LIN {X 0,Y 466.068,Z 1064.204,A -85,B 0,C 180,E1 20747.984,E2 20747.984} C_VEL
LIN {X 0,Y 471.463,Z 1046.564,A -85,B 0,C 180,E1 20746.009,E2 20746.009} C_VEL
LIN {X 0,Y 478.479,Z 1022.709,A -85,B 0,C 180,E1 20743.696,E2 20743.696} C_VEL
LIN {X 0,Y 484.027,Z 1002.948,A -85,B 0,C 180,E1 20742.045,E2 20742.045} C_VEL
LIN {X 0,Y 489.037,Z 984.19,A -85,B 0,C 180,E1 20740.666,E2 20740.666} C_VEL
LIN {X 0,Y 494.055,Z 964.129,A -85,B 0,C 180,E1 20739.369,E2 20739.369} C_VEL
LIN {X 0,Y 500.021,Z 937.929,A -85,B 0,C 180,E1 20737.922,E2 20737.922} C_VEL
LIN {X 0,Y 504.618,Z 915.146,A -85,B 0,C 180,E1 20736.878,E2 20736.878} C_VEL
LIN {X 0,Y 508.385,Z 894.221,A -85,B 0,C 180,E1 20736.067,E2 20736.067} C_VEL
LIN {X 0,Y 511.805,Z 872.432,A -85,B 0,C 180,E1 20735.363,E2 20735.363} C_VEL
LIN {X 0,Y 515.371,Z 845.255,A -85,B 0,C 180,E1 20734.667,E2 20734.667} C_VEL
LIN {X 0,Y 517.719,Z 818.939,A -85,B 0,C 180,E1 20734.166,E2 20734.166} C_VEL
LIN {X 0,Y 527.517,Z 618.648,A -85,B 0,C 180,E1 20731.083,E2 20731.083} C_VEL
LIN {X 0,Y 535.309,Z 463.056,A -85,B 0,C 180,E1 20728.673,E2 20728.673} C_VEL
LIN {X 0,Y 522.466,Z 443.048,A -85,B 0,C 180,E1 20726.054,E2 20726.054} C_VEL
LIN {X 0,Y 512.066,Z 427.582,A -85,B 0,C 180,E1 20723.719,E2 20723.719} C_VEL
LIN {X 0,Y 502.428,Z 413.843,A -85,B 0,C 180,E1 20721.327,E2 20721.327} C_VEL
LIN {X 0,Y 493.826,Z 402.221,A -85,B 0,C 180,E1 20718.964,E2 20718.964} C_VEL
LIN {X 0,Y 487.693,Z 394.13,A -85,B 0,C 180,E1 20717.11,E2 20717.11} C_VEL
LIN {X 0,Y 479.768,Z 384.005,A -85,B 0,C 180,E1 20714.421,E2 20714.421} C_VEL
LIN {X 0,Y 474.951,Z 378.127,A -85,B 0,C 180,E1 20712.585,E2 20712.585} C_VEL
LIN {X 0,Y 471.073,Z 373.273,A -85,B 0,C 180,E1 20710.951,E2 20710.951} C_VEL
LIN {X 0,Y 466.248,Z 367.542,A -85,B 0,C 180,E1 20708.66,E2 20708.66} C_VEL
LIN {X 0,Y 460.499,Z 361.075,A -85,B 0,C 180,E1 20705.357,E2 20705.357} C_VEL
LIN {X 0,Y 456.273,Z 356.326,A -85,B 0,C 180,E1 20702.21,E2 20702.21} C_VEL
LIN {X 0,Y 455.002,Z 354.829,A -85,B 0,C 180,E1 20701.007,E2 20701.007} C_VEL
LIN {X 0,Y 451.289,Z 351.259,A -85,B 0,C 180,E1 20695.17,E2 20695.17} C_VEL
LIN {X 0,Y 451.06,Z 350.914,A -85,B 0,C 180,E1 20691.972,E2 20691.972} C_VEL
LIN {X 0,Y 452.202,Z 352.442,A -85,B 0,C 180,E1 20688.133,E2 20688.133} C_VEL
LIN {X 0,Y 455.623,Z 355.438,A -85,B 0,C 180,E1 20683.948,E2 20683.948} C_VEL
LIN {X 0,Y 459.701,Z 360.404,A -85,B 0,C 180,E1 20680.694,E2 20680.694} C_VEL
LIN {X 0,Y 461.444,Z 362.203,A -85,B 0,C 180,E1 20679.582,E2 20679.582} C_VEL
LIN {X 0,Y 465.451,Z 366.813,A -85,B 0,C 180,E1 20677.319,E2 20677.319} C_VEL
LIN {X 0,Y 471.187,Z 373.665,A -85,B 0,C 180,E1 20674.55,E2 20674.55} C_VEL
LIN {X 0,Y 476.082,Z 379.677,A -85,B 0,C 180,E1 20672.514,E2 20672.514} C_VEL
LIN {X 0,Y 480.917,Z 385.697,A -85,B 0,C 180,E1 20670.717,E2 20670.717} C_VEL
LIN {X 0,Y 487.922,Z 394.605,A -85,B 0,C 180,E1 20668.392,E2 20668.392} C_VEL
LIN {X 0,Y 496.453,Z 405.98,A -85,B 0,C 180,E1 20665.88,E2 20665.88} C_VEL
LIN {X 0,Y 506.01,Z 419.292,A -85,B 0,C 180,E1 20663.362,E2 20663.362} C_VEL
LIN {X 0,Y 516.742,Z 435.021,A -85,B 0,C 180,E1 20660.819,E2 20660.819} C_VEL
LIN {X 0,Y 528.945,Z 454.078,A -85,B 0,C 180,E1 20658.214,E2 20658.214} C_VEL
LIN {X 0,Y 530.531,Z 456.882,A -85,B 0,C 180,E1 20657.888,E2 20657.888} C_VEL
LIN {X 0,Y 518.704,Z 687.315,A -85,B 0,C 180,E1 20654.4,E2 20654.4} C_VEL
LIN {X 0,Y 513.437,Z 790.124,A -85,B 0,C 180,E1 20652.825,E2 20652.825} C_VEL
LIN {X 0,Y 510.977,Z 817.179,A -85,B 0,C 180,E1 20652.266,E2 20652.266} C_VEL
LIN {X 0,Y 507.981,Z 840.872,A -85,B 0,C 180,E1 20651.597,E2 20651.597} C_VEL
LIN {X 0,Y 504.867,Z 861.286,A -85,B 0,C 180,E1 20650.884,E2 20650.884} C_VEL
LIN {X 0,Y 500.818,Z 884.029,A -85,B 0,C 180,E1 20649.93,E2 20649.93} C_VEL
LIN {X 0,Y 495.731,Z 908.011,A -85,B 0,C 180,E1 20648.7,E2 20648.7} C_VEL
LIN {X 0,Y 491.245,Z 926.964,A -85,B 0,C 180,E1 20647.56,E2 20647.56} C_VEL
LIN {X 0,Y 486.131,Z 946.852,A -85,B 0,C 180,E1 20646.178,E2 20646.178} C_VEL
LIN {X 0,Y 479.73,Z 969.616,A -85,B 0,C 180,E1 20644.317,E2 20644.317} C_VEL
LIN {X 0,Y 474.426,Z 987.14,A -85,B 0,C 180,E1 20642.651,E2 20642.651} C_VEL
LIN {X 0,Y 468.964,Z 1004.442,A -85,B 0,C 180,E1 20640.777,E2 20640.777} C_VEL
LIN {X 0,Y 462.391,Z 1024.359,A -85,B 0,C 180,E1 20638.265,E2 20638.265} C_VEL
LIN {X 0,Y 457.591,Z 1038.554,A -85,B 0,C 180,E1 20636.192,E2 20636.192} C_VEL
LIN {X 0,Y 453.023,Z 1052.055,A -85,B 0,C 180,E1 20633.96,E2 20633.96} C_VEL
LIN {X 0,Y 452.093,Z 1054.945,A -85,B 0,C 180,E1 20633.456,E2 20633.456} C_VEL
LIN {X 0,Y 449.768,Z 1059.456,A -85,B 0,C 180,E1 20632.709,E2 20632.709} C_VEL
LIN {X 0,Y 440.278,Z 1071.251,A -85,B 0,C 180,E1 20630.787,E2 20630.787} C_VEL
LIN {X 0,Y 438.47,Z 1074.724,A -85,B 0,C 180,E1 20630.085,E2 20630.085} C_VEL
LIN {X 0,Y 434.176,Z 1087.706,A -85,B 0,C 180,E1 20626.868,E2 20626.868} C_VEL
LIN {X 0,Y 431.232,Z 1097.26,A -85,B 0,C 180,E1 20624.09,E2 20624.09} C_VEL
LIN {X 0,Y 428.732,Z 1106.306,A -85,B 0,C 180,E1 20621.025,E2 20621.025} C_VEL
LIN {X 0,Y 426.702,Z 1114.7,A -85,B 0,C 180,E1 20617.54,E2 20617.54} C_VEL
LIN {X 0,Y 425.561,Z 1120.466,A -85,B 0,C 180,E1 20614.582,E2 20614.582} C_VEL
LIN {X 0,Y 424.864,Z 1124.898,A -85,B 0,C 180,E1 20611.753,E2 20611.753} C_VEL
LIN {X 0,Y 424.443,Z 1128.897,A -85,B 0,C 180,E1 20608.38,E2 20608.38} C_VEL
LIN {X 0,Y 424.242,Z 1131.291,A -85,B 0,C 180,E1 20604.997,E2 20604.997} C_VEL
LIN {X 0,Y 424.216,Z 1132.271,A -85,B 0,C 180,E1 20602.143,E2 20602.143} C_VEL
LIN {X 0,Y 424.205,Z 1132.282,A -85,B 0,C 180,E1 20599.393,E2 20599.393} C_VEL
LIN {X 0,Y 424.282,Z 1131.313,A -85,B 0,C 180,E1 20596.508,E2 20596.508} C_VEL
LIN {X 0,Y 424.543,Z 1128.64,A -85,B 0,C 180,E1 20592.879,E2 20592.879} C_VEL
LIN {X 0,Y 425.024,Z 1125,A -85,B 0,C 180,E1 20589.768,E2 20589.768} C_VEL
LIN {X 0,Y 425.805,Z 1120.621,A -85,B 0,C 180,E1 20586.912,E2 20586.912} C_VEL
LIN {X 0,Y 427.274,Z 1114.277,A -85,B 0,C 180,E1 20583.601,E2 20583.601} C_VEL
LIN {X 0,Y 429.569,Z 1105.855,A -85,B 0,C 180,E1 20580.125,E2 20580.125} C_VEL
LIN {X 0,Y 432.214,Z 1097.455,A -85,B 0,C 180,E1 20577.226,E2 20577.226} C_VEL
LIN {X 0,Y 435.991,Z 1086.706,A -85,B 0,C 180,E1 20574.05,E2 20574.05} C_VEL
LIN {X 0,Y 440.717,Z 1073.903,A -85,B 0,C 180,E1 20570.889,E2 20570.889} C_VEL
LIN {X 0,Y 445.319,Z 1062.002,A -85,B 0,C 180,E1 20568.349,E2 20568.349} C_VEL
LIN {X 0,Y 451.443,Z 1046.625,A -85,B 0,C 180,E1 20565.495,E2 20565.495} C_VEL
LIN {X 0,Y 457.914,Z 1030.027,A -85,B 0,C 180,E1 20562.898,E2 20562.898} C_VEL
LIN {X 0,Y 463.585,Z 1015.355,A -85,B 0,C 180,E1 20560.891,E2 20560.891} C_VEL
LIN {X 0,Y 470.718,Z 996.54,A -85,B 0,C 180,E1 20558.646,E2 20558.646} C_VEL
LIN {X 0,Y 477.551,Z 977.158,A -85,B 0,C 180,E1 20556.689,E2 20556.689} C_VEL
LIN {X 0,Y 483.256,Z 960.126,A -85,B 0,C 180,E1 20555.189,E2 20555.189} C_VEL
LIN {X 0,Y 488.91,Z 942.119,A -85,B 0,C 180,E1 20553.799,E2 20553.799} C_VEL
LIN {X 0,Y 495.538,Z 919.171,A -85,B 0,C 180,E1 20552.282,E2 20552.282} C_VEL
LIN {X 0,Y 500.941,Z 897.811,A -85,B 0,C 180,E1 20551.1,E2 20551.1} C_VEL
LIN {X 0,Y 505.444,Z 877.923,A -85,B 0,C 180,E1 20550.164,E2 20550.164} C_VEL
LIN {X 0,Y 509.85,Z 855.684,A -85,B 0,C 180,E1 20549.286,E2 20549.286} C_VEL
LIN {X 0,Y 514.128,Z 828.821,A -85,B 0,C 180,E1 20548.445,E2 20548.445} C_VEL
LIN {X 0,Y 516.842,Z 807.129,A -85,B 0,C 180,E1 20547.926,E2 20547.926} C_VEL
LIN {X 0,Y 518.863,Z 784.756,A -85,B 0,C 180,E1 20547.509,E2 20547.509} C_VEL
LIN {X 0,Y 533.637,Z 545.962,A -85,B 0,C 180,E1 20543.837,E2 20543.837} C_VEL
LIN {X 0,Y 538.73,Z 467.206,A -85,B 0,C 180,E1 20542.63,E2 20542.63} C_VEL
LIN {X 0,Y 531.191,Z 455.254,A -85,B 0,C 180,E1 20540.495,E2 20540.495} C_VEL
LIN {X 0,Y 523.295,Z 443.397,A -85,B 0,C 180,E1 20537.974,E2 20537.974} C_VEL
LIN {X 0,Y 516.807,Z 434.328,A -85,B 0,C 180,E1 20535.601,E2 20535.601} C_VEL
LIN {X 0,Y 512.914,Z 428.986,A -85,B 0,C 180,E1 20533.989,E2 20533.989} C_VEL
LIN {X 0,Y 509.266,Z 424.025,A -85,B 0,C 180,E1 20532.3,E2 20532.3} C_VEL
LIN {X 0,Y 505.818,Z 419.487,A -85,B 0,C 180,E1 20530.478,E2 20530.478} C_VEL
LIN {X 0,Y 502.428,Z 414.973,A -85,B 0,C 180,E1 20528.353,E2 20528.353} C_VEL
LIN {X 0,Y 498.483,Z 409.718,A -85,B 0,C 180,E1 20525.063,E2 20525.063} C_VEL
LIN {X 0,Y 495.085,Z 405.672,A -85,B 0,C 180,E1 20519.421,E2 20519.421} C_VEL
LIN {X 0,Y 495.033,Z 405.551,A -85,B 0,C 180,E1 20516.642,E2 20516.642} C_VEL
LIN {X 0,Y 496.724,Z 408.094,A -85,B 0,C 180,E1 20512.714,E2 20512.714} C_VEL
LIN {X 0,Y 499.227,Z 410.598,A -85,B 0,C 180,E1 20509.965,E2 20509.965} C_VEL
LIN {X 0,Y 503.669,Z 416.542,A -85,B 0,C 180,E1 20506.569,E2 20506.569} C_VEL
LIN {X 0,Y 507.835,Z 422.101,A -85,B 0,C 180,E1 20504.175,E2 20504.175} C_VEL
LIN {X 0,Y 511.462,Z 426.885,A -85,B 0,C 180,E1 20502.42,E2 20502.42} C_VEL
LIN {X 0,Y 515.737,Z 432.762,A -85,B 0,C 180,E1 20500.579,E2 20500.579} C_VEL
LIN {X 0,Y 520.757,Z 439.738,A -85,B 0,C 180,E1 20498.663,E2 20498.663} C_VEL
LIN {X 0,Y 527.808,Z 450.043,A -85,B 0,C 180,E1 20496.291,E2 20496.291} C_VEL
LIN {X 0,Y 535.871,Z 462.538,A -85,B 0,C 180,E1 20493.903,E2 20493.903} C_VEL
LIN {X 0,Y 540.756,Z 470.818,A -85,B 0,C 180,E1 20492.572,E2 20492.572} C_VEL
LIN {X 0,Y 527.788,Z 678.066,A -85,B 0,C 180,E1 20489.301,E2 20489.301} C_VEL
LIN {X 0,Y 519.327,Z 818.255,A -85,B 0,C 180,E1 20487.08,E2 20487.08} C_VEL
LIN {X 0,Y 516.4,Z 846.054,A -85,B 0,C 180,E1 20486.538,E2 20486.538} C_VEL
LIN {X 0,Y 512.544,Z 871.525,A -85,B 0,C 180,E1 20485.88,E2 20485.88} C_VEL
LIN {X 0,Y 508.877,Z 892.088,A -85,B 0,C 180,E1 20485.215,E2 20485.215} C_VEL
LIN {X 0,Y 504.658,Z 912.7,A -85,B 0,C 180,E1 20484.42,E2 20484.42} C_VEL
LIN {X 0,Y 499.778,Z 934.113,A -85,B 0,C 180,E1 20483.441,E2 20483.441} C_VEL
LIN {X 0,Y 493.02,Z 960.613,A -85,B 0,C 180,E1 20481.989,E2 20481.989} C_VEL
LIN {X 0,Y 487.098,Z 981.501,A -85,B 0,C 180,E1 20480.632,E2 20480.632} C_VEL
LIN {X 0,Y 481.367,Z 1000.582,A -85,B 0,C 180,E1 20479.21,E2 20479.21} C_VEL
LIN {X 0,Y 475.341,Z 1019.687,A -85,B 0,C 180,E1 20477.588,E2 20477.588} C_VEL
LIN {X 0,Y 467.897,Z 1042.428,A -85,B 0,C 180,E1 20475.365,E2 20475.365} C_VEL
LIN {X 0,Y 461.269,Z 1061.82,A -85,B 0,C 180,E1 20473.152,E2 20473.152} C_VEL
LIN {X 0,Y 455.592,Z 1078.396,A -85,B 0,C 180,E1 20471.01,E2 20471.01} C_VEL
LIN {X 0,Y 450.042,Z 1094.732,A -85,B 0,C 180,E1 20468.631,E2 20468.631} C_VEL
LIN {X 0,Y 443.578,Z 1114.036,A -85,B 0,C 180,E1 20465.401,E2 20465.401} C_VEL
LIN {X 0,Y 439.042,Z 1128.205,A -85,B 0,C 180,E1 20462.666,E2 20462.666} C_VEL
LIN {X 0,Y 435.408,Z 1140.323,A -85,B 0,C 180,E1 20460.03,E2 20460.03} C_VEL
LIN {X 0,Y 431.826,Z 1153.297,A -85,B 0,C 180,E1 20456.84,E2 20456.84} C_VEL
LIN {X 0,Y 428.772,Z 1165.845,A -85,B 0,C 180,E1 20453.209,E2 20453.209} C_VEL
LIN {X 0,Y 426.968,Z 1174.525,A -85,B 0,C 180,E1 20450.278,E2 20450.278} C_VEL
LIN {X 0,Y 425.739,Z 1181.638,A -85,B 0,C 180,E1 20447.494,E2 20447.494} C_VEL
LIN {X 0,Y 424.919,Z 1187.651,A -85,B 0,C 180,E1 20444.722,E2 20444.722} C_VEL
LIN {X 0,Y 424.406,Z 1192.596,A -85,B 0,C 180,E1 20441.965,E2 20441.965} C_VEL
LIN {X 0,Y 424.144,Z 1196.504,A -85,B 0,C 180,E1 20439.224,E2 20439.224} C_VEL
LIN {X 0,Y 424.039,Z 1199.394,A -85,B 0,C 180,E1 20436.499,E2 20436.499} C_VEL
LIN {X 0,Y 424.011,Z 1201.284,A -85,B 0,C 180,E1 20433.786,E2 20433.786} C_VEL
LIN {X 0,Y 424.015,Z 1202.183,A -85,B 0,C 180,E1 20431.081,E2 20431.081} C_VEL
LIN {X 0,Y 424.015,Z 1202.119,A -85,B 0,C 180,E1 20428.514,E2 20428.514} C_VEL
LIN {X 0,Y 424.01,Z 1201.166,A -85,B 0,C 180,E1 20425.943,E2 20425.943} C_VEL
LIN {X 0,Y 424.037,Z 1199.324,A -85,B 0,C 180,E1 20423.365,E2 20423.365} C_VEL
LIN {X 0,Y 424.149,Z 1196.412,A -85,B 0,C 180,E1 20420.639,E2 20420.639} C_VEL
LIN {X 0,Y 424.424,Z 1192.456,A -85,B 0,C 180,E1 20417.876,E2 20417.876} C_VEL
LIN {X 0,Y 424.949,Z 1187.536,A -85,B 0,C 180,E1 20415.14,E2 20415.14} C_VEL
LIN {X 0,Y 425.834,Z 1181.193,A -85,B 0,C 180,E1 20412.228,E2 20412.228} C_VEL
LIN {X 0,Y 427.351,Z 1172.886,A -85,B 0,C 180,E1 20409.025,E2 20409.025} C_VEL
LIN {X 0,Y 429.839,Z 1161.535,A -85,B 0,C 180,E1 20405.394,E2 20405.394} C_VEL
LIN {X 0,Y 432.543,Z 1150.782,A -85,B 0,C 180,E1 20402.464,E2 20402.464} C_VEL
LIN {X 0,Y 435.609,Z 1139.765,A -85,B 0,C 180,E1 20399.823,E2 20399.823} C_VEL
LIN {X 0,Y 439.354,Z 1127.015,A -85,B 0,C 180,E1 20397.117,E2 20397.117} C_VEL
LIN {X 0,Y 444.791,Z 1109.649,A -85,B 0,C 180,E1 20393.917,E2 20393.917} C_VEL
LIN {X 0,Y 449.903,Z 1093.567,A -85,B 0,C 180,E1 20391.355,E2 20391.355} C_VEL
LIN {X 0,Y 454.732,Z 1078.539,A -85,B 0,C 180,E1 20389.229,E2 20389.229} C_VEL
LIN {X 0,Y 460.057,Z 1061.94,A -85,B 0,C 180,E1 20387.137,E2 20387.137} C_VEL
LIN {X 0,Y 466.809,Z 1040.494,A -85,B 0,C 180,E1 20384.771,E2 20384.771} C_VEL
LIN {X 0,Y 472.997,Z 1019.875,A -85,B 0,C 180,E1 20382.818,E2 20382.818} C_VEL
LIN {X 0,Y 478.368,Z 1001.288,A -85,B 0,C 180,E1 20381.273,E2 20381.273} C_VEL
LIN {X 0,Y 483.974,Z 980.835,A -85,B 0,C 180,E1 20379.778,E2 20379.778} C_VEL
LIN {X 0,Y 490.636,Z 954.332,A -85,B 0,C 180,E1 20378.129,E2 20378.129} C_VEL
LIN {X 0,Y 495.364,Z 933.437,A -85,B 0,C 180,E1 20377.033,E2 20377.033} C_VEL
LIN {X 0,Y 499.614,Z 912.696,A -85,B 0,C 180,E1 20376.098,E2 20376.098} C_VEL
LIN {X 0,Y 503.486,Z 891.607,A -85,B 0,C 180,E1 20375.295,E2 20375.295} C_VEL
LIN {X 0,Y 507.68,Z 865.101,A -85,B 0,C 180,E1 20374.466,E2 20374.466} C_VEL
LIN {X 0,Y 510.906,Z 838.43,A -85,B 0,C 180,E1 20373.842,E2 20373.842} C_VEL
LIN {X 0,Y 512.827,Z 815.961,A -85,B 0,C 180,E1 20373.427,E2 20373.427} C_VEL
LIN {X 0,Y 523.598,Z 602.198,A -85,B 0,C 180,E1 20370.124,E2 20370.124} C_VEL
LIN {X 0,Y 530.557,Z 467.247,A -85,B 0,C 180,E1 20368.017,E2 20368.017} C_VEL
LIN {X 0,Y 518.234,Z 447.75,A -85,B 0,C 180,E1 20365.423,E2 20365.423} C_VEL
LIN {X 0,Y 506.469,Z 430.195,A -85,B 0,C 180,E1 20362.673,E2 20362.673} C_VEL
LIN {X 0,Y 496.569,Z 416.22,A -85,B 0,C 180,E1 20360.079,E2 20360.079} C_VEL
LIN {X 0,Y 488.595,Z 405.412,A -85,B 0,C 180,E1 20357.754,E2 20357.754} C_VEL
LIN {X 0,Y 481.271,Z 395.879,A -85,B 0,C 180,E1 20355.361,E2 20355.361} C_VEL
LIN {X 0,Y 477.499,Z 391.017,A -85,B 0,C 180,E1 20353.996,E2 20353.996} C_VEL
LIN {X 0,Y 473.213,Z 385.642,A -85,B 0,C 180,E1 20352.322,E2 20352.322} C_VEL
LIN {X 0,Y 468.342,Z 379.691,A -85,B 0,C 180,E1 20350.207,E2 20350.207} C_VEL
LIN {X 0,Y 463.914,Z 374.392,A -85,B 0,C 180,E1 20347.991,E2 20347.991} C_VEL
LIN {X 0,Y 459.316,Z 368.937,A -85,B 0,C 180,E1 20345.246,E2 20345.246} C_VEL
LIN {X 0,Y 455.061,Z 364.08,A -85,B 0,C 180,E1 20342.015,E2 20342.015} C_VEL
LIN {X 0,Y 453.892,Z 362.701,A -85,B 0,C 180,E1 20340.884,E2 20340.884} C_VEL
LIN {X 0,Y 450.282,Z 359.154,A -85,B 0,C 180,E1 20335.032,E2 20335.032} C_VEL
LIN {X 0,Y 450.098,Z 358.875,A -85,B 0,C 180,E1 20331.826,E2 20331.826} C_VEL
LIN {X 0,Y 451.46,Z 360.644,A -85,B 0,C 180,E1 20327.724,E2 20327.724} C_VEL
LIN {X 0,Y 454.536,Z 363.358,A -85,B 0,C 180,E1 20324.039,E2 20324.039} C_VEL
LIN {X 0,Y 458.39,Z 368.148,A -85,B 0,C 180,E1 20320.901,E2 20320.901} C_VEL
LIN {X 0,Y 460.105,Z 369.923,A -85,B 0,C 180,E1 20319.785,E2 20319.785} C_VEL
LIN {X 0,Y 464.166,Z 374.636,A -85,B 0,C 180,E1 20317.453,E2 20317.453} C_VEL
LIN {X 0,Y 469.719,Z 381.458,A -85,B 0,C 180,E1 20314.735,E2 20314.735} C_VEL
LIN {X 0,Y 474.412,Z 387.293,A -85,B 0,C 180,E1 20312.749,E2 20312.749} C_VEL
LIN {X 0,Y 479.079,Z 393.185,A -85,B 0,C 180,E1 20310.982,E2 20310.982} C_VEL
LIN {X 0,Y 485.845,Z 401.923,A -85,B 0,C 180,E1 20308.691,E2 20308.691} C_VEL
LIN {X 0,Y 494.169,Z 413.181,A -85,B 0,C 180,E1 20306.191,E2 20306.191} C_VEL
LIN {X 0,Y 503.51,Z 426.378,A -85,B 0,C 180,E1 20303.681,E2 20303.681} C_VEL
LIN {X 0,Y 513.899,Z 441.801,A -85,B 0,C 180,E1 20301.171,E2 20301.171} C_VEL
LIN {X 0,Y 525.903,Z 460.797,A -85,B 0,C 180,E1 20298.556,E2 20298.556} C_VEL
LIN {X 0,Y 513.733,Z 690.618,A -85,B 0,C 180,E1 20295.063,E2 20295.063} C_VEL
LIN {X 0,Y 508.459,Z 790.477,A -85,B 0,C 180,E1 20293.526,E2 20293.526} C_VEL
LIN {X 0,Y 505.934,Z 817.545,A -85,B 0,C 180,E1 20292.966,E2 20292.966} C_VEL
LIN {X 0,Y 502.887,Z 841.077,A -85,B 0,C 180,E1 20292.3,E2 20292.3} C_VEL
LIN {X 0,Y 499.82,Z 860.714,A -85,B 0,C 180,E1 20291.617,E2 20291.617} C_VEL
LIN {X 0,Y 496.089,Z 881.182,A -85,B 0,C 180,E1 20290.769,E2 20290.769} C_VEL
LIN {X 0,Y 490.647,Z 906.855,A -85,B 0,C 180,E1 20289.48,E2 20289.48} C_VEL
LIN {X 0,Y 485.799,Z 926.857,A -85,B 0,C 180,E1 20288.28,E2 20288.28} C_VEL
LIN {X 0,Y 480.719,Z 946.05,A -85,B 0,C 180,E1 20286.948,E2 20286.948} C_VEL
LIN {X 0,Y 474.181,Z 968.82,A -85,B 0,C 180,E1 20285.098,E2 20285.098} C_VEL
LIN {X 0,Y 468.43,Z 987.272,A -85,B 0,C 180,E1 20283.342,E2 20283.342} C_VEL
LIN {X 0,Y 463.053,Z 1003.748,A -85,B 0,C 180,E1 20281.553,E2 20281.553} C_VEL
LIN {X 0,Y 456.755,Z 1022.44,A -85,B 0,C 180,E1 20279.219,E2 20279.219} C_VEL
LIN {X 0,Y 451.111,Z 1038.46,A -85,B 0,C 180,E1 20276.882,E2 20276.882} C_VEL
LIN {X 0,Y 446.33,Z 1052.031,A -85,B 0,C 180,E1 20274.625,E2 20274.625} C_VEL
LIN {X 0,Y 441.222,Z 1066.792,A -85,B 0,C 180,E1 20271.817,E2 20271.817} C_VEL
LIN {X 0,Y 438.47,Z 1074.724,A -85,B 0,C 180,E1 20270.085,E2 20270.085} C_VEL
LIN {X 0,Y 436.293,Z 1078.674,A -85,B 0,C 180,E1 20269.257,E2 20269.257} C_VEL
LIN {X 0,Y 427.62,Z 1088.44,A -85,B 0,C 180,E1 20267.22,E2 20267.22} C_VEL
LIN {X 0,Y 425.602,Z 1091.898,A -85,B 0,C 180,E1 20266.327,E2 20266.327} C_VEL
LIN {X 0,Y 422.087,Z 1103.225,A -85,B 0,C 180,E1 20262.727,E2 20262.727} C_VEL
LIN {X 0,Y 419.933,Z 1111.038,A -85,B 0,C 180,E1 20259.733,E2 20259.733} C_VEL
LIN {X 0,Y 418.339,Z 1117.903,A -85,B 0,C 180,E1 20256.588,E2 20256.588} C_VEL
LIN {X 0,Y 417.154,Z 1124.218,A -85,B 0,C 180,E1 20252.885,E2 20252.885} C_VEL
LIN {X 0,Y 416.612,Z 1128.07,A -85,B 0,C 180,E1 20249.862,E2 20249.862} C_VEL
LIN {X 0,Y 416.362,Z 1130.622,A -85,B 0,C 180,E1 20247.109,E2 20247.109} C_VEL
LIN {X 0,Y 416.256,Z 1132.338,A -85,B 0,C 180,E1 20244.21,E2 20244.21} C_VEL
LIN {X 0,Y 416.235,Z 1133.14,A -85,B 0,C 180,E1 20240.738,E2 20240.738} C_VEL
LIN {X 0,Y 416.29,Z 1132.407,A -85,B 0,C 180,E1 20237.375,E2 20237.375} C_VEL
LIN {X 0,Y 416.412,Z 1130.819,A -85,B 0,C 180,E1 20234.542,E2 20234.542} C_VEL
LIN {X 0,Y 416.731,Z 1128.265,A -85,B 0,C 180,E1 20231.681,E2 20231.681} C_VEL
LIN {X 0,Y 417.378,Z 1124.317,A -85,B 0,C 180,E1 20228.499,E2 20228.499} C_VEL
LIN {X 0,Y 418.792,Z 1117.9,A -85,B 0,C 180,E1 20224.7,E2 20224.7} C_VEL
LIN {X 0,Y 420.469,Z 1111.653,A -85,B 0,C 180,E1 20221.757,E2 20221.757} C_VEL
LIN {X 0,Y 422.793,Z 1104.21,A -85,B 0,C 180,E1 20218.808,E2 20218.808} C_VEL
LIN {X 0,Y 426.694,Z 1093.049,A -85,B 0,C 180,E1 20215.127,E2 20215.127} C_VEL
LIN {X 0,Y 430.707,Z 1082.44,A -85,B 0,C 180,E1 20212.203,E2 20212.203} C_VEL
LIN {X 0,Y 435.289,Z 1070.944,A -85,B 0,C 180,E1 20209.455,E2 20209.455} C_VEL
LIN {X 0,Y 441.838,Z 1054.97,A -85,B 0,C 180,E1 20206.212,E2 20206.212} C_VEL
LIN {X 0,Y 447.539,Z 1041.122,A -85,B 0,C 180,E1 20203.811,E2 20203.811} C_VEL
LIN {X 0,Y 453.822,Z 1025.791,A -85,B 0,C 180,E1 20201.489,E2 20201.489} C_VEL
LIN {X 0,Y 461.575,Z 1006.174,A -85,B 0,C 180,E1 20198.953,E2 20198.953} C_VEL
LIN {X 0,Y 467.795,Z 989.775,A -85,B 0,C 180,E1 20197.132,E2 20197.132} C_VEL
LIN {X 0,Y 474.439,Z 971.433,A -85,B 0,C 180,E1 20195.355,E2 20195.355} C_VEL
LIN {X 0,Y 482,Z 948.814,A -85,B 0,C 180,E1 20193.491,E2 20193.491} C_VEL
LIN {X 0,Y 487.802,Z 929.852,A -85,B 0,C 180,E1 20192.163,E2 20192.163} C_VEL
LIN {X 0,Y 493.296,Z 910.247,A -85,B 0,C 180,E1 20190.977,E2 20190.977} C_VEL
LIN {X 0,Y 499.242,Z 886.515,A -85,B 0,C 180,E1 20189.762,E2 20189.762} C_VEL
LIN {X 0,Y 503.969,Z 864.133,A -85,B 0,C 180,E1 20188.824,E2 20188.824} C_VEL
LIN {X 0,Y 507.554,Z 844.352,A -85,B 0,C 180,E1 20188.132,E2 20188.132} C_VEL
LIN {X 0,Y 510.841,Z 822.463,A -85,B 0,C 180,E1 20187.504,E2 20187.504} C_VEL
LIN {X 0,Y 514.053,Z 794.047,A -85,B 0,C 180,E1 20186.899,E2 20186.899} C_VEL
LIN {X 0,Y 518.149,Z 731.579,A -85,B 0,C 180,E1 20185.916,E2 20185.916} C_VEL
LIN {X 0,Y 533.591,Z 492.448,A -85,B 0,C 180,E1 20182.242,E2 20182.242} C_VEL
LIN {X 0,Y 534.953,Z 471.915,A -85,B 0,C 180,E1 20181.923,E2 20181.923} C_VEL
LIN {X 0,Y 527.585,Z 460.132,A -85,B 0,C 180,E1 20179.744,E2 20179.744} C_VEL
LIN {X 0,Y 519.175,Z 447.481,A -85,B 0,C 180,E1 20176.907,E2 20176.907} C_VEL
LIN {X 0,Y 512.179,Z 437.573,A -85,B 0,C 180,E1 20174.125,E2 20174.125} C_VEL
LIN {X 0,Y 507.723,Z 431.572,A -85,B 0,C 180,E1 20172.049,E2 20172.049} C_VEL
LIN {X 0,Y 504.443,Z 427.168,A -85,B 0,C 180,E1 20170.276,E2 20170.276} C_VEL
LIN {X 0,Y 501.284,Z 422.847,A -85,B 0,C 180,E1 20168.257,E2 20168.257} C_VEL
LIN {X 0,Y 497.384,Z 417.595,A -85,B 0,C 180,E1 20164.959,E2 20164.959} C_VEL
LIN {X 0,Y 494.106,Z 413.62,A -85,B 0,C 180,E1 20159.42,E2 20159.42} C_VEL
LIN {X 0,Y 494.038,Z 413.463,A -85,B 0,C 180,E1 20156.751,E2 20156.751} C_VEL
LIN {X 0,Y 495.58,Z 415.883,A -85,B 0,C 180,E1 20152.93,E2 20152.93} C_VEL
LIN {X 0,Y 498.118,Z 418.514,A -85,B 0,C 180,E1 20150.059,E2 20150.059} C_VEL
LIN {X 0,Y 502.425,Z 424.37,A -85,B 0,C 180,E1 20146.711,E2 20146.711} C_VEL
LIN {X 0,Y 506.42,Z 429.807,A -85,B 0,C 180,E1 20144.365,E2 20144.365} C_VEL
LIN {X 0,Y 509.987,Z 434.622,A -85,B 0,C 180,E1 20142.603,E2 20142.603} C_VEL
LIN {X 0,Y 514.337,Z 440.708,A -85,B 0,C 180,E1 20140.702,E2 20140.702} C_VEL
LIN {X 0,Y 519.395,Z 447.789,A -85,B 0,C 180,E1 20138.752,E2 20138.752} C_VEL
LIN {X 0,Y 526.871,Z 459.109,A -85,B 0,C 180,E1 20136.216,E2 20136.216} C_VEL
LIN {X 0,Y 534.212,Z 470.736,A -85,B 0,C 180,E1 20134.025,E2 20134.025} C_VEL
LIN {X 0,Y 536.907,Z 475.544,A -85,B 0,C 180,E1 20133.265,E2 20133.265} C_VEL
LIN {X 0,Y 523.457,Z 684.035,A -85,B 0,C 180,E1 20129.969,E2 20129.969} C_VEL
LIN {X 0,Y 515.115,Z 817.846,A -85,B 0,C 180,E1 20127.842,E2 20127.842} C_VEL
LIN {X 0,Y 512.103,Z 845.678,A -85,B 0,C 180,E1 20127.3,E2 20127.3} C_VEL
LIN {X 0,Y 508.148,Z 871.138,A -85,B 0,C 180,E1 20126.644,E2 20126.644} C_VEL
LIN {X 0,Y 504.308,Z 892.059,A -85,B 0,C 180,E1 20125.97,E2 20125.97} C_VEL
LIN {X 0,Y 499.98,Z 912.611,A -85,B 0,C 180,E1 20125.177,E2 20125.177} C_VEL
LIN {X 0,Y 494.687,Z 935.078,A -85,B 0,C 180,E1 20124.145,E2 20124.145} C_VEL
LIN {X 0,Y 487.729,Z 961.249,A -85,B 0,C 180,E1 20122.694,E2 20122.694} C_VEL
LIN {X 0,Y 481.843,Z 981.352,A -85,B 0,C 180,E1 20121.382,E2 20121.382} C_VEL
LIN {X 0,Y 475.736,Z 1000.967,A -85,B 0,C 180,E1 20119.909,E2 20119.909} C_VEL
LIN {X 0,Y 468.853,Z 1022.012,A -85,B 0,C 180,E1 20118.096,E2 20118.096} C_VEL
LIN {X 0,Y 460.988,Z 1044.808,A -85,B 0,C 180,E1 20115.794,E2 20115.794} C_VEL
LIN {X 0,Y 454.728,Z 1062.444,A -85,B 0,C 180,E1 20113.742,E2 20113.742} C_VEL
LIN {X 0,Y 448.871,Z 1078.816,A -85,B 0,C 180,E1 20111.59,E2 20111.59} C_VEL
LIN {X 0,Y 442.239,Z 1097.676,A -85,B 0,C 180,E1 20108.775,E2 20108.775} C_VEL
LIN {X 0,Y 436.082,Z 1115.08,A -85,B 0,C 180,E1 20105.739,E2 20105.739} C_VEL
LIN {X 0,Y 431.673,Z 1128.233,A -85,B 0,C 180,E1 20103.136,E2 20103.136} C_VEL
LIN {X 0,Y 427.725,Z 1140.84,A -85,B 0,C 180,E1 20100.326,E2 20100.326} C_VEL
LIN {X 0,Y 423.602,Z 1155.188,A -85,B 0,C 180,E1 20096.646,E2 20096.646} C_VEL
LIN {X 0,Y 420.861,Z 1166.01,A -85,B 0,C 180,E1 20093.375,E2 20093.375} C_VEL
LIN {X 0,Y 419.08,Z 1174.191,A -85,B 0,C 180,E1 20090.531,E2 20090.531} C_VEL
LIN {X 0,Y 417.798,Z 1181.246,A -85,B 0,C 180,E1 20087.694,E2 20087.694} C_VEL
LIN {X 0,Y 416.919,Z 1187.491,A -85,B 0,C 180,E1 20084.727,E2 20084.727} C_VEL
LIN {X 0,Y 416.343,Z 1193.02,A -85,B 0,C 180,E1 20081.498,E2 20081.498} C_VEL
LIN {X 0,Y 416.095,Z 1197.596,A -85,B 0,C 180,E1 20077.873,E2 20077.873} C_VEL
LIN {X 0,Y 416.04,Z 1200.168,A -85,B 0,C 180,E1 20074.687,E2 20074.687} C_VEL
LIN {X 0,Y 416.04,Z 1201.396,A -85,B 0,C 180,E1 20071.79,E2 20071.79} C_VEL
LIN {X 0,Y 416.038,Z 1201.557,A -85,B 0,C 180,E1 20069.036,E2 20069.036} C_VEL
LIN {X 0,Y 416.033,Z 1200.729,A -85,B 0,C 180,E1 20066.28,E2 20066.28} C_VEL
LIN {X 0,Y 416.055,Z 1198.909,A -85,B 0,C 180,E1 20063.515,E2 20063.515} C_VEL
LIN {X 0,Y 416.154,Z 1196.09,A -85,B 0,C 180,E1 20060.737,E2 20060.737} C_VEL
LIN {X 0,Y 416.439,Z 1192.038,A -85,B 0,C 180,E1 20057.802,E2 20057.802} C_VEL
LIN {X 0,Y 416.982,Z 1187.123,A -85,B 0,C 180,E1 20054.991,E2 20054.991} C_VEL
LIN {X 0,Y 417.848,Z 1181.138,A -85,B 0,C 180,E1 20052.164,E2 20052.164} C_VEL
LIN {X 0,Y 419.161,Z 1174.046,A -85,B 0,C 180,E1 20049.327,E2 20049.327} C_VEL
LIN {X 0,Y 421.08,Z 1165.358,A -85,B 0,C 180,E1 20046.341,E2 20046.341} C_VEL
LIN {X 0,Y 424.301,Z 1152.695,A -85,B 0,C 180,E1 20042.644,E2 20042.644} C_VEL
LIN {X 0,Y 427.83,Z 1140.347,A -85,B 0,C 180,E1 20039.587,E2 20039.587} C_VEL
LIN {X 0,Y 431.427,Z 1128.501,A -85,B 0,C 180,E1 20037.001,E2 20037.001} C_VEL
LIN {X 0,Y 435.561,Z 1115.591,A -85,B 0,C 180,E1 20034.495,E2 20034.495} C_VEL
LIN {X 0,Y 441.188,Z 1098.762,A -85,B 0,C 180,E1 20031.614,E2 20031.614} C_VEL
LIN {X 0,Y 447.385,Z 1080.023,A -85,B 0,C 180,E1 20028.867,E2 20028.867} C_VEL
LIN {X 0,Y 452.727,Z 1063.934,A -85,B 0,C 180,E1 20026.789,E2 20026.789} C_VEL
LIN {X 0,Y 458.287,Z 1046.962,A -85,B 0,C 180,E1 20024.842,E2 20024.842} C_VEL
LIN {X 0,Y 465.132,Z 1025.497,A -85,B 0,C 180,E1 20022.679,E2 20022.679} C_VEL
LIN {X 0,Y 471.866,Z 1002.885,A -85,B 0,C 180,E1 20020.742,E2 20020.742} C_VEL
LIN {X 0,Y 477.148,Z 984.317,A -85,B 0,C 180,E1 20019.355,E2 20019.355} C_VEL
LIN {X 0,Y 482.194,Z 965.386,A -85,B 0,C 180,E1 20018.11,E2 20018.11} C_VEL
LIN {X 0,Y 487.728,Z 942.857,A -85,B 0,C 180,E1 20016.819,E2 20016.819} C_VEL
LIN {X 0,Y 493.536,Z 916.18,A -85,B 0,C 180,E1 20015.553,E2 20015.553} C_VEL
LIN {X 0,Y 497.703,Z 894.37,A -85,B 0,C 180,E1 20014.699,E2 20014.699} C_VEL
LIN {X 0,Y 501.256,Z 872.965,A -85,B 0,C 180,E1 20013.999,E2 20013.999} C_VEL
LIN {X 0,Y 504.724,Z 848.321,A -85,B 0,C 180,E1 20013.353,E2 20013.353} C_VEL
LIN {X 0,Y 507.548,Z 819.795,A -85,B 0,C 180,E1 20012.789,E2 20012.789} C_VEL
LIN {X 0,Y 512.531,Z 725.573,A -85,B 0,C 180,E1 20011.313,E2 20011.313} C_VEL
LIN {X 0,Y 524.181,Z 504.486,A -85,B 0,C 180,E1 20007.887,E2 20007.887} C_VEL
LIN {X 0,Y 525.871,Z 471.383,A -85,B 0,C 180,E1 20007.352,E2 20007.352} C_VEL
LIN {X 0,Y 514.38,Z 453.099,A -85,B 0,C 180,E1 20004.858,E2 20004.858} C_VEL
LIN {X 0,Y 503.552,Z 436.725,A -85,B 0,C 180,E1 20002.257,E2 20002.257} C_VEL
LIN {X 0,Y 494.087,Z 423.176,A -85,B 0,C 180,E1 19999.722,E2 19999.722} C_VEL
LIN {X 0,Y 486.32,Z 412.501,A -85,B 0,C 180,E1 19997.407,E2 19997.407} C_VEL
LIN {X 0,Y 478.957,Z 402.797,A -85,B 0,C 180,E1 19994.941,E2 19994.941} C_VEL
LIN {X 0,Y 475.405,Z 398.179,A -85,B 0,C 180,E1 19993.625,E2 19993.625} C_VEL
LIN {X 0,Y 471.485,Z 393.155,A -85,B 0,C 180,E1 19992.057,E2 19992.057} C_VEL
LIN {X 0,Y 466.567,Z 387.077,A -85,B 0,C 180,E1 19989.872,E2 19989.872} C_VEL
LIN {X 0,Y 462.462,Z 382.062,A -85,B 0,C 180,E1 19987.766,E2 19987.766} C_VEL
LIN {X 0,Y 457.942,Z 376.641,A -85,B 0,C 180,E1 19985.01,E2 19985.01} C_VEL
LIN {X 0,Y 453.674,Z 371.553,A -85,B 0,C 180,E1 19981.642,E2 19981.642} C_VEL
LIN {X 0,Y 452.067,Z 370.043,A -85,B 0,C 180,E1 19980,E2 19980} C_VEL
LIN {X 0,Y 449.249,Z 367.006,A -85,B 0,C 180,E1 19974.764,E2 19974.764} C_VEL
LIN {X 0,Y 449.154,Z 366.854,A -85,B 0,C 180,E1 19971.551,E2 19971.551} C_VEL
LIN {X 0,Y 450.824,Z 368.927,A -85,B 0,C 180,E1 19967.186,E2 19967.186} C_VEL
LIN {X 0,Y 453.451,Z 371.277,A -85,B 0,C 180,E1 19964.132,E2 19964.132} C_VEL
LIN {X 0,Y 457.269,Z 376.049,A -85,B 0,C 180,E1 19960.985,E2 19960.985} C_VEL
LIN {X 0,Y 458.865,Z 377.784,A -85,B 0,C 180,E1 19959.928,E2 19959.928} C_VEL
LIN {X 0,Y 463.667,Z 383.599,A -85,B 0,C 180,E1 19957.159,E2 19957.159} C_VEL
LIN {X 0,Y 468.129,Z 389.05,A -85,B 0,C 180,E1 19954.981,E2 19954.981} C_VEL
LIN {X 0,Y 472.679,Z 394.801,A -85,B 0,C 180,E1 19953.016,E2 19953.016} C_VEL
LIN {X 0,Y 477.303,Z 400.743,A -85,B 0,C 180,E1 19951.23,E2 19951.23} C_VEL
LIN {X 0,Y 483.782,Z 409.239,A -85,B 0,C 180,E1 19948.992,E2 19948.992} C_VEL
LIN {X 0,Y 491.9,Z 420.379,A -85,B 0,C 180,E1 19946.504,E2 19946.504} C_VEL
LIN {X 0,Y 501.026,Z 433.462,A -85,B 0,C 180,E1 19944.004,E2 19944.004} C_VEL
LIN {X 0,Y 511.196,Z 448.792,A -85,B 0,C 180,E1 19941.498,E2 19941.498} C_VEL
LIN {X 0,Y 521.328,Z 465.014,A -85,B 0,C 180,E1 19939.231,E2 19939.231} C_VEL
LIN {X 0,Y 508.768,Z 695.05,A -85,B 0,C 180,E1 19935.722,E2 19935.722} C_VEL
LIN {X 0,Y 503.529,Z 791.005,A -85,B 0,C 180,E1 19934.237,E2 19934.237} C_VEL
LIN {X 0,Y 500.899,Z 818.351,A -85,B 0,C 180,E1 19933.667,E2 19933.667} C_VEL
LIN {X 0,Y 497.796,Z 841.714,A -85,B 0,C 180,E1 19933.004,E2 19933.004} C_VEL
LIN {X 0,Y 494.616,Z 861.537,A -85,B 0,C 180,E1 19932.311,E2 19932.311} C_VEL
LIN {X 0,Y 490.33,Z 884.386,A -85,B 0,C 180,E1 19931.352,E2 19931.352} C_VEL
LIN {X 0,Y 484.938,Z 908.618,A -85,B 0,C 180,E1 19930.107,E2 19930.107} C_VEL
LIN {X 0,Y 480.206,Z 927.555,A -85,B 0,C 180,E1 19928.962,E2 19928.962} C_VEL
LIN {X 0,Y 474.984,Z 946.753,A -85,B 0,C 180,E1 19927.623,E2 19927.623} C_VEL
LIN {X 0,Y 467.971,Z 970.372,A -85,B 0,C 180,E1 19925.682,E2 19925.682} C_VEL
LIN {X 0,Y 462.312,Z 987.954,A -85,B 0,C 180,E1 19923.991,E2 19923.991} C_VEL
LIN {X 0,Y 456.641,Z 1004.79,A -85,B 0,C 180,E1 19922.145,E2 19922.145} C_VEL
LIN {X 0,Y 449.595,Z 1024.86,A -85,B 0,C 180,E1 19919.584,E2 19919.584} C_VEL
LIN {X 0,Y 444.107,Z 1039.928,A -85,B 0,C 180,E1 19917.341,E2 19917.341} C_VEL
LIN {X 0,Y 439.031,Z 1053.837,A -85,B 0,C 180,E1 19914.981,E2 19914.981} C_VEL
LIN {X 0,Y 433.226,Z 1069.842,A -85,B 0,C 180,E1 19911.813,E2 19911.813} C_VEL
LIN {X 0,Y 429.19,Z 1081.21,A -85,B 0,C 180,E1 19909.176,E2 19909.176} C_VEL
LIN {X 0,Y 425.652,Z 1091.737,A -85,B 0,C 180,E1 19906.372,E2 19906.372} C_VEL
LIN {X 0,Y 425.602,Z 1091.898,A -85,B 0,C 180,E1 19906.327,E2 19906.327} C_VEL
LIN {X 0,Y 423.643,Z 1095.264,A -85,B 0,C 180,E1 19905.42,E2 19905.42} C_VEL
LIN {X 0,Y 415.143,Z 1103.95,A -85,B 0,C 180,E1 19903.034,E2 19903.034} C_VEL
LIN {X 0,Y 413.715,Z 1106.361,A -85,B 0,C 180,E1 19902.2,E2 19902.2} C_VEL
LIN {X 0,Y 411.382,Z 1114.917,A -85,B 0,C 180,E1 19898.667,E2 19898.667} C_VEL
LIN {X 0,Y 409.899,Z 1121.325,A -85,B 0,C 180,E1 19895.318,E2 19895.318} C_VEL
LIN {X 0,Y 409.09,Z 1125.836,A -85,B 0,C 180,E1 19892.381,E2 19892.381} C_VEL
LIN {X 0,Y 408.578,Z 1129.625,A -85,B 0,C 180,E1 19889.159,E2 19889.159} C_VEL
LIN {X 0,Y 408.314,Z 1132.412,A -85,B 0,C 180,E1 19885.506,E2 19885.506} C_VEL
LIN {X 0,Y 408.262,Z 1133.541,A -85,B 0,C 180,E1 19882.4,E2 19882.4} C_VEL
LIN {X 0,Y 408.262,Z 1133.642,A -85,B 0,C 180,E1 19879.558,E2 19879.558} C_VEL
LIN {X 0,Y 408.337,Z 1132.826,A -85,B 0,C 180,E1 19876.693,E2 19876.693} C_VEL
LIN {X 0,Y 408.537,Z 1130.946,A -85,B 0,C 180,E1 19873.622,E2 19873.622} C_VEL
LIN {X 0,Y 409.129,Z 1127.095,A -85,B 0,C 180,E1 19869.798,E2 19869.798} C_VEL
LIN {X 0,Y 410.059,Z 1122.498,A -85,B 0,C 180,E1 19866.581,E2 19866.581} C_VEL
LIN {X 0,Y 411.424,Z 1117.151,A -85,B 0,C 180,E1 19863.594,E2 19863.594} C_VEL
LIN {X 0,Y 413.871,Z 1109.288,A -85,B 0,C 180,E1 19859.994,E2 19859.994} C_VEL
LIN {X 0,Y 417.141,Z 1099.806,A -85,B 0,C 180,E1 19856.529,E2 19856.529} C_VEL
LIN {X 0,Y 420.635,Z 1090.715,A -85,B 0,C 180,E1 19853.691,E2 19853.691} C_VEL
LIN {X 0,Y 425.727,Z 1078.385,A -85,B 0,C 180,E1 19850.387,E2 19850.387} C_VEL
LIN {X 0,Y 431.323,Z 1065.044,A -85,B 0,C 180,E1 19847.399,E2 19847.399} C_VEL
LIN {X 0,Y 436.69,Z 1052.569,A -85,B 0,C 180,E1 19844.968,E2 19844.968} C_VEL
LIN {X 0,Y 443.669,Z 1036.479,A -85,B 0,C 180,E1 19842.242,E2 19842.242} C_VEL
LIN {X 0,Y 451.048,Z 1018.773,A -85,B 0,C 180,E1 19839.717,E2 19839.717} C_VEL
LIN {X 0,Y 457.367,Z 1003.22,A -85,B 0,C 180,E1 19837.788,E2 19837.788} C_VEL
LIN {X 0,Y 464.894,Z 984.018,A -85,B 0,C 180,E1 19835.718,E2 19835.718} C_VEL
LIN {X 0,Y 472.374,Z 963.216,A -85,B 0,C 180,E1 19833.828,E2 19833.828} C_VEL
LIN {X 0,Y 478.181,Z 945.935,A -85,B 0,C 180,E1 19832.467,E2 19832.467} C_VEL
LIN {X 0,Y 484.212,Z 926.554,A -85,B 0,C 180,E1 19831.14,E2 19831.14} C_VEL
LIN {X 0,Y 491.336,Z 900.854,A -85,B 0,C 180,E1 19829.665,E2 19829.665} C_VEL
LIN {X 0,Y 496.356,Z 879.988,A -85,B 0,C 180,E1 19828.673,E2 19828.673} C_VEL
LIN {X 0,Y 500.843,Z 858.663,A -85,B 0,C 180,E1 19827.824,E2 19827.824} C_VEL
LIN {X 0,Y 505.43,Z 832.165,A -85,B 0,C 180,E1 19826.976,E2 19826.976} C_VEL
LIN {X 0,Y 508.479,Z 809.296,A -85,B 0,C 180,E1 19826.42,E2 19826.42} C_VEL
LIN {X 0,Y 510.577,Z 787.809,A -85,B 0,C 180,E1 19826.012,E2 19826.012} C_VEL
LIN {X 0,Y 526.124,Z 552.076,A -85,B 0,C 180,E1 19822.372,E2 19822.372} C_VEL
LIN {X 0,Y 531.24,Z 476.677,A -85,B 0,C 180,E1 19821.203,E2 19821.203} C_VEL
LIN {X 0,Y 524.769,Z 466.317,A -85,B 0,C 180,E1 19819.218,E2 19819.218} C_VEL
LIN {X 0,Y 517.305,Z 454.827,A -85,B 0,C 180,E1 19816.623,E2 19816.623} C_VEL
LIN {X 0,Y 510.435,Z 444.958,A -85,B 0,C 180,E1 19813.827,E2 19813.827} C_VEL
LIN {X 0,Y 506.192,Z 439.115,A -85,B 0,C 180,E1 19811.797,E2 19811.797} C_VEL
LIN {X 0,Y 502.98,Z 434.732,A -85,B 0,C 180,E1 19810.017,E2 19810.017} C_VEL
LIN {X 0,Y 499.978,Z 430.567,A -85,B 0,C 180,E1 19808.047,E2 19808.047} C_VEL
LIN {X 0,Y 496.286,Z 425.473,A -85,B 0,C 180,E1 19804.854,E2 19804.854} C_VEL
LIN {X 0,Y 493.103,Z 421.519,A -85,B 0,C 180,E1 19799.303,E2 19799.303} C_VEL
LIN {X 0,Y 493.077,Z 421.445,A -85,B 0,C 180,E1 19796.629,E2 19796.629} C_VEL
LIN {X 0,Y 494.925,Z 424.234,A -85,B 0,C 180,E1 19792.454,E2 19792.454} C_VEL
LIN {X 0,Y 496.955,Z 426.323,A -85,B 0,C 180,E1 19790.211,E2 19790.211} C_VEL
LIN {X 0,Y 501.101,Z 432.065,A -85,B 0,C 180,E1 19786.91,E2 19786.91} C_VEL
LIN {X 0,Y 505.016,Z 437.512,A -85,B 0,C 180,E1 19784.556,E2 19784.556} C_VEL
LIN {X 0,Y 508.403,Z 442.175,A -85,B 0,C 180,E1 19782.842,E2 19782.842} C_VEL
LIN {X 0,Y 512.554,Z 448.077,A -85,B 0,C 180,E1 19780.987,E2 19780.987} C_VEL
LIN {X 0,Y 517.594,Z 455.286,A -85,B 0,C 180,E1 19779.001,E2 19779.001} C_VEL
LIN {X 0,Y 525.042,Z 466.749,A -85,B 0,C 180,E1 19776.426,E2 19776.426} C_VEL
LIN {X 0,Y 532.648,Z 479.058,A -85,B 0,C 180,E1 19774.122,E2 19774.122} C_VEL
LIN {X 0,Y 533.148,Z 480.257,A -85,B 0,C 180,E1 19773.968,E2 19773.968} C_VEL
LIN {X 0,Y 519.174,Z 690.662,A -85,B 0,C 180,E1 19770.638,E2 19770.638} C_VEL
LIN {X 0,Y 510.996,Z 817.548,A -85,B 0,C 180,E1 19768.616,E2 19768.616} C_VEL
LIN {X 0,Y 507.88,Z 845.544,A -85,B 0,C 180,E1 19768.069,E2 19768.069} C_VEL
LIN {X 0,Y 503.889,Z 870.613,A -85,B 0,C 180,E1 19767.426,E2 19767.426} C_VEL
LIN {X 0,Y 500.075,Z 890.866,A -85,B 0,C 180,E1 19766.78,E2 19766.78} C_VEL
LIN {X 0,Y 495.684,Z 911.241,A -85,B 0,C 180,E1 19766,E2 19766} C_VEL
LIN {X 0,Y 490.506,Z 932.672,A -85,B 0,C 180,E1 19765.029,E2 19765.029} C_VEL
LIN {X 0,Y 483.327,Z 959.205,A -85,B 0,C 180,E1 19763.584,E2 19763.584} C_VEL
LIN {X 0,Y 476.709,Z 981.105,A -85,B 0,C 180,E1 19762.156,E2 19762.156} C_VEL
LIN {X 0,Y 470.544,Z 1000.3,A -85,B 0,C 180,E1 19760.71,E2 19760.71} C_VEL
LIN {X 0,Y 463.774,Z 1020.28,A -85,B 0,C 180,E1 19758.988,E2 19758.988} C_VEL
LIN {X 0,Y 455.363,Z 1043.809,A -85,B 0,C 180,E1 19756.618,E2 19756.618} C_VEL
LIN {X 0,Y 448.733,Z 1061.754,A -85,B 0,C 180,E1 19754.517,E2 19754.517} C_VEL
LIN {X 0,Y 442.552,Z 1078.315,A -85,B 0,C 180,E1 19752.32,E2 19752.32} C_VEL
LIN {X 0,Y 435.631,Z 1097.121,A -85,B 0,C 180,E1 19749.477,E2 19749.477} C_VEL
LIN {X 0,Y 429.277,Z 1114.313,A -85,B 0,C 180,E1 19746.437,E2 19746.437} C_VEL
LIN {X 0,Y 424.562,Z 1127.64,A -85,B 0,C 180,E1 19743.761,E2 19743.761} C_VEL
LIN {X 0,Y 420.594,Z 1139.599,A -85,B 0,C 180,E1 19741.055,E2 19741.055} C_VEL
LIN {X 0,Y 416.349,Z 1153.552,A -85,B 0,C 180,E1 19737.457,E2 19737.457} C_VEL
LIN {X 0,Y 413.276,Z 1164.9,A -85,B 0,C 180,E1 19733.982,E2 19733.982} C_VEL
LIN {X 0,Y 411.279,Z 1173.504,A -85,B 0,C 180,E1 19730.939,E2 19730.939} C_VEL
LIN {X 0,Y 409.913,Z 1180.552,A -85,B 0,C 180,E1 19728.046,E2 19728.046} C_VEL
LIN {X 0,Y 408.986,Z 1186.795,A -85,B 0,C 180,E1 19725.019,E2 19725.019} C_VEL
LIN {X 0,Y 408.37,Z 1192.446,A -85,B 0,C 180,E1 19721.65,E2 19721.65} C_VEL
LIN {X 0,Y 408.118,Z 1196.92,A -85,B 0,C 180,E1 19718.027,E2 19718.027} C_VEL
LIN {X 0,Y 408.066,Z 1199.503,A -85,B 0,C 180,E1 19714.779,E2 19714.779} C_VEL
LIN {X 0,Y 408.067,Z 1200.737,A -85,B 0,C 180,E1 19711.825,E2 19711.825} C_VEL
LIN {X 0,Y 408.066,Z 1200.901,A -85,B 0,C 180,E1 19709.017,E2 19709.017} C_VEL
LIN {X 0,Y 408.057,Z 1200.073,A -85,B 0,C 180,E1 19706.207,E2 19706.207} C_VEL
LIN {X 0,Y 408.074,Z 1198.249,A -85,B 0,C 180,E1 19703.387,E2 19703.387} C_VEL
LIN {X 0,Y 408.18,Z 1195.424,A -85,B 0,C 180,E1 19700.554,E2 19700.554} C_VEL
LIN {X 0,Y 408.469,Z 1191.438,A -85,B 0,C 180,E1 19697.612,E2 19697.612} C_VEL
LIN {X 0,Y 409.055,Z 1186.425,A -85,B 0,C 180,E1 19694.693,E2 19694.693} C_VEL
LIN {X 0,Y 409.969,Z 1180.413,A -85,B 0,C 180,E1 19691.81,E2 19691.81} C_VEL
LIN {X 0,Y 411.365,Z 1173.29,A -85,B 0,C 180,E1 19688.917,E2 19688.917} C_VEL
LIN {X 0,Y 413.502,Z 1164.131,A -85,B 0,C 180,E1 19685.728,E2 19685.728} C_VEL
LIN {X 0,Y 416.978,Z 1151.189,A -85,B 0,C 180,E1 19681.939,E2 19681.939} C_VEL
LIN {X 0,Y 420.383,Z 1139.813,A -85,B 0,C 180,E1 19679.087,E2 19679.087} C_VEL
LIN {X 0,Y 424.052,Z 1128.236,A -85,B 0,C 180,E1 19676.514,E2 19676.514} C_VEL
LIN {X 0,Y 428.356,Z 1115.337,A -85,B 0,C 180,E1 19673.97,E2 19673.97} C_VEL
LIN {X 0,Y 434.192,Z 1098.539,A -85,B 0,C 180,E1 19671.048,E2 19671.048} C_VEL
LIN {X 0,Y 440.654,Z 1079.68,A -85,B 0,C 180,E1 19668.244,E2 19668.244} C_VEL
LIN {X 0,Y 446.117,Z 1063.81,A -85,B 0,C 180,E1 19666.168,E2 19666.168} C_VEL
LIN {X 0,Y 451.869,Z 1046.833,A -85,B 0,C 180,E1 19664.199,E2 19664.199} C_VEL
LIN {X 0,Y 458.928,Z 1025.438,A -85,B 0,C 180,E1 19662.019,E2 19662.019} C_VEL
LIN {X 0,Y 465.788,Z 1003.136,A -85,B 0,C 180,E1 19660.091,E2 19660.091} C_VEL
LIN {X 0,Y 471.536,Z 983.487,A -85,B 0,C 180,E1 19658.613,E2 19658.613} C_VEL
LIN {X 0,Y 476.763,Z 964.456,A -85,B 0,C 180,E1 19657.361,E2 19657.361} C_VEL
LIN {X 0,Y 482.704,Z 940.89,A -85,B 0,C 180,E1 19656.015,E2 19656.015} C_VEL
LIN {X 0,Y 488.349,Z 915.355,A -85,B 0,C 180,E1 19654.814,E2 19654.814} C_VEL
LIN {X 0,Y 492.54,Z 894.005,A -85,B 0,C 180,E1 19653.978,E2 19653.978} C_VEL
LIN {X 0,Y 496.179,Z 872.618,A -85,B 0,C 180,E1 19653.278,E2 19653.278} C_VEL
LIN {X 0,Y 499.71,Z 848.148,A -85,B 0,C 180,E1 19652.636,E2 19652.636} C_VEL
LIN {X 0,Y 502.615,Z 819.535,A -85,B 0,C 180,E1 19652.068,E2 19652.068} C_VEL
LIN {X 0,Y 507.666,Z 726.915,A -85,B 0,C 180,E1 19650.611,E2 19650.611} C_VEL
LIN {X 0,Y 519.687,Z 505.853,A -85,B 0,C 180,E1 19647.172,E2 19647.172} C_VEL
LIN {X 0,Y 521.365,Z 475.647,A -85,B 0,C 180,E1 19646.696,E2 19646.696} C_VEL
LIN {X 0,Y 509.082,Z 455.982,A -85,B 0,C 180,E1 19643.928,E2 19643.928} C_VEL
LIN {X 0,Y 497.282,Z 438.217,A -85,B 0,C 180,E1 19640.941,E2 19640.941} C_VEL
LIN {X 0,Y 488.315,Z 425.428,A -85,B 0,C 180,E1 19638.381,E2 19638.381} C_VEL
LIN {X 0,Y 481.102,Z 415.528,A -85,B 0,C 180,E1 19636.078,E2 19636.078} C_VEL
LIN {X 0,Y 473.783,Z 405.849,A -85,B 0,C 180,E1 19633.424,E2 19633.424} C_VEL
LIN {X 0,Y 469.625,Z 400.522,A -85,B 0,C 180,E1 19631.732,E2 19631.732} C_VEL
LIN {X 0,Y 464.933,Z 394.596,A -85,B 0,C 180,E1 19629.594,E2 19629.594} C_VEL
LIN {X 0,Y 461.015,Z 389.731,A -85,B 0,C 180,E1 19627.54,E2 19627.54} C_VEL
LIN {X 0,Y 456.575,Z 384.345,A -85,B 0,C 180,E1 19624.774,E2 19624.774} C_VEL
LIN {X 0,Y 451.802,Z 378.535,A -85,B 0,C 180,E1 19620.761,E2 19620.761} C_VEL
LIN {X 0,Y 448.301,Z 374.995,A -85,B 0,C 180,E1 19614.881,E2 19614.881} C_VEL
LIN {X 0,Y 448.147,Z 374.762,A -85,B 0,C 180,E1 19611.79,E2 19611.79} C_VEL
LIN {X 0,Y 449.544,Z 376.59,A -85,B 0,C 180,E1 19607.671,E2 19607.671} C_VEL
LIN {X 0,Y 452.245,Z 379.002,A -85,B 0,C 180,E1 19604.351,E2 19604.351} C_VEL
LIN {X 0,Y 456.149,Z 383.949,A -85,B 0,C 180,E1 19601.069,E2 19601.069} C_VEL
LIN {X 0,Y 457.628,Z 385.643,A -85,B 0,C 180,E1 19600.071,E2 19600.071} C_VEL
LIN {X 0,Y 462.258,Z 391.337,A -85,B 0,C 180,E1 19597.355,E2 19597.355} C_VEL
LIN {X 0,Y 466.411,Z 396.45,A -85,B 0,C 180,E1 19595.289,E2 19595.289} C_VEL
LIN {X 0,Y 470.957,Z 402.307,A -85,B 0,C 180,E1 19593.284,E2 19593.284} C_VEL
LIN {X 0,Y 475.512,Z 408.26,A -85,B 0,C 180,E1 19591.489,E2 19591.489} C_VEL
LIN {X 0,Y 481.733,Z 416.552,A -85,B 0,C 180,E1 19589.296,E2 19589.296} C_VEL
LIN {X 0,Y 489.74,Z 427.714,A -85,B 0,C 180,E1 19586.792,E2 19586.792} C_VEL
LIN {X 0,Y 498.453,Z 440.39,A -85,B 0,C 180,E1 19584.356,E2 19584.356} C_VEL
LIN {X 0,Y 508.378,Z 455.57,A -85,B 0,C 180,E1 19581.86,E2 19581.86} C_VEL
LIN {X 0,Y 516.821,Z 469.332,A -85,B 0,C 180,E1 19579.915,E2 19579.915} C_VEL
LIN {X 0,Y 503.747,Z 701.688,A -85,B 0,C 180,E1 19576.36,E2 19576.36} C_VEL
LIN {X 0,Y 498.685,Z 791.446,A -85,B 0,C 180,E1 19574.964,E2 19574.964} C_VEL
LIN {X 0,Y 495.973,Z 818.883,A -85,B 0,C 180,E1 19574.39,E2 19574.39} C_VEL
LIN {X 0,Y 492.804,Z 842.146,A -85,B 0,C 180,E1 19573.727,E2 19573.727} C_VEL
LIN {X 0,Y 489.603,Z 861.605,A -85,B 0,C 180,E1 19573.047,E2 19573.047} C_VEL
LIN {X 0,Y 485.406,Z 883.452,A -85,B 0,C 180,E1 19572.135,E2 19572.135} C_VEL
LIN {X 0,Y 479.806,Z 908.285,A -85,B 0,C 180,E1 19570.869,E2 19570.869} C_VEL
LIN {X 0,Y 474.685,Z 928.255,A -85,B 0,C 180,E1 19569.66,E2 19569.66} C_VEL
LIN {X 0,Y 469.099,Z 948.202,A -85,B 0,C 180,E1 19568.256,E2 19568.256} C_VEL
LIN {X 0,Y 462.088,Z 971.041,A -85,B 0,C 180,E1 19566.361,E2 19566.361} C_VEL
LIN {X 0,Y 456.256,Z 988.634,A -85,B 0,C 180,E1 19564.658,E2 19564.658} C_VEL
LIN {X 0,Y 450.402,Z 1005.465,A -85,B 0,C 180,E1 19562.797,E2 19562.797} C_VEL
LIN {X 0,Y 443.072,Z 1025.64,A -85,B 0,C 180,E1 19560.194,E2 19560.194} C_VEL
LIN {X 0,Y 437.434,Z 1040.604,A -85,B 0,C 180,E1 19557.942,E2 19557.942} C_VEL
LIN {X 0,Y 432.046,Z 1054.826,A -85,B 0,C 180,E1 19555.496,E2 19555.496} C_VEL
LIN {X 0,Y 426.114,Z 1070.513,A -85,B 0,C 180,E1 19552.341,E2 19552.341} C_VEL
LIN {X 0,Y 421.911,Z 1081.886,A -85,B 0,C 180,E1 19549.665,E2 19549.665} C_VEL
LIN {X 0,Y 418.202,Z 1092.408,A -85,B 0,C 180,E1 19546.815,E2 19546.815} C_VEL
LIN {X 0,Y 414.462,Z 1103.896,A -85,B 0,C 180,E1 19543.107,E2 19543.107} C_VEL
LIN {X 0,Y 413.715,Z 1106.361,A -85,B 0,C 180,E1 19542.2,E2 19542.2} C_VEL
LIN {X 0,Y 411.994,Z 1109.156,A -85,B 0,C 180,E1 19541.221,E2 19541.221} C_VEL
LIN {X 0,Y 404.146,Z 1116.18,A -85,B 0,C 180,E1 19538.625,E2 19538.625} C_VEL
LIN {X 0,Y 402.955,Z 1118.038,A -85,B 0,C 180,E1 19537.734,E2 19537.734} C_VEL
LIN {X 0,Y 401.623,Z 1124.111,A -85,B 0,C 180,E1 19534.283,E2 19534.283} C_VEL
LIN {X 0,Y 400.791,Z 1128.937,A -85,B 0,C 180,E1 19530.572,E2 19530.572} C_VEL
LIN {X 0,Y 400.461,Z 1131.719,A -85,B 0,C 180,E1 19527.567,E2 19527.567} C_VEL
LIN {X 0,Y 400.319,Z 1133.453,A -85,B 0,C 180,E1 19524.697,E2 19524.697} C_VEL
LIN {X 0,Y 400.295,Z 1134.291,A -85,B 0,C 180,E1 19521.815,E2 19521.815} C_VEL
LIN {X 0,Y 400.318,Z 1134.177,A -85,B 0,C 180,E1 19518.474,E2 19518.474} C_VEL
LIN {X 0,Y 400.469,Z 1132.583,A -85,B 0,C 180,E1 19514.802,E2 19514.802} C_VEL
LIN {X 0,Y 400.822,Z 1130.073,A -85,B 0,C 180,E1 19511.681,E2 19511.681} C_VEL
LIN {X 0,Y 401.44,Z 1126.673,A -85,B 0,C 180,E1 19508.676,E2 19508.676} C_VEL
LIN {X 0,Y 402.567,Z 1121.99,A -85,B 0,C 180,E1 19505.495,E2 19505.495} C_VEL
LIN {X 0,Y 404.791,Z 1114.466,A -85,B 0,C 180,E1 19501.528,E2 19501.528} C_VEL
LIN {X 0,Y 407.409,Z 1106.87,A -85,B 0,C 180,E1 19498.318,E2 19498.318} C_VEL
LIN {X 0,Y 410.678,Z 1098.356,A -85,B 0,C 180,E1 19495.27,E2 19495.27} C_VEL
LIN {X 0,Y 415.943,Z 1085.713,A -85,B 0,C 180,E1 19491.494,E2 19491.494} C_VEL
LIN {X 0,Y 420.85,Z 1074.431,A -85,B 0,C 180,E1 19488.658,E2 19488.658} C_VEL
LIN {X 0,Y 426.768,Z 1061.293,A -85,B 0,C 180,E1 19485.803,E2 19485.803} C_VEL
LIN {X 0,Y 434.077,Z 1045.004,A -85,B 0,C 180,E1 19482.807,E2 19482.807} C_VEL
LIN {X 0,Y 440.327,Z 1030.883,A -85,B 0,C 180,E1 19480.575,E2 19480.575} C_VEL
LIN {X 0,Y 446.976,Z 1015.551,A -85,B 0,C 180,E1 19478.454,E2 19478.454} C_VEL
LIN {X 0,Y 455.405,Z 995.217,A -85,B 0,C 180,E1 19476.045,E2 19476.045} C_VEL
LIN {X 0,Y 462.234,Z 977.688,A -85,B 0,C 180,E1 19474.279,E2 19474.279} C_VEL
LIN {X 0,Y 468.529,Z 960.573,A -85,B 0,C 180,E1 19472.774,E2 19472.774} C_VEL
LIN {X 0,Y 475.116,Z 941.369,A -85,B 0,C 180,E1 19471.306,E2 19471.306} C_VEL
LIN {X 0,Y 482.537,Z 917.188,A -85,B 0,C 180,E1 19469.749,E2 19469.749} C_VEL
LIN {X 0,Y 487.85,Z 897.757,A -85,B 0,C 180,E1 19468.694,E2 19468.694} C_VEL
LIN {X 0,Y 492.843,Z 877.209,A -85,B 0,C 180,E1 19467.743,E2 19467.743} C_VEL
LIN {X 0,Y 498.26,Z 850.998,A -85,B 0,C 180,E1 19466.75,E2 19466.75} C_VEL
LIN {X 0,Y 502.088,Z 827.672,A -85,B 0,C 180,E1 19466.055,E2 19466.055} C_VEL
LIN {X 0,Y 504.989,Z 805.639,A -85,B 0,C 180,E1 19465.547,E2 19465.547} C_VEL
LIN {X 0,Y 507.562,Z 776.631,A -85,B 0,C 180,E1 19465.038,E2 19465.038} C_VEL
LIN {X 0,Y 523.699,Z 538.021,A -85,B 0,C 180,E1 19461.36,E2 19461.36} C_VEL
LIN {X 0,Y 527.683,Z 481.575,A -85,B 0,C 180,E1 19460.492,E2 19460.492} C_VEL
LIN {X 0,Y 520.174,Z 469.489,A -85,B 0,C 180,E1 19458.057,E2 19458.057} C_VEL
LIN {X 0,Y 513.99,Z 460.141,A -85,B 0,C 180,E1 19455.775,E2 19455.775} C_VEL
LIN {X 0,Y 508.222,Z 451.728,A -85,B 0,C 180,E1 19453.308,E2 19453.308} C_VEL
LIN {X 0,Y 504.671,Z 446.658,A -85,B 0,C 180,E1 19451.543,E2 19451.543} C_VEL
LIN {X 0,Y 501.62,Z 442.412,A -85,B 0,C 180,E1 19449.813,E2 19449.813} C_VEL
LIN {X 0,Y 498.678,Z 438.284,A -85,B 0,C 180,E1 19447.836,E2 19447.836} C_VEL
LIN {X 0,Y 495.191,Z 433.35,A -85,B 0,C 180,E1 19444.749,E2 19444.749} C_VEL
LIN {X 0,Y 492.124,Z 429.467,A -85,B 0,C 180,E1 19439.302,E2 19439.302} C_VEL
LIN {X 0,Y 492.099,Z 429.393,A -85,B 0,C 180,E1 19436.622,E2 19436.622} C_VEL
LIN {X 0,Y 494.03,Z 432.303,A -85,B 0,C 180,E1 19432.323,E2 19432.323} C_VEL
LIN {X 0,Y 495.848,Z 434.243,A -85,B 0,C 180,E1 19430.306,E2 19430.306} C_VEL
LIN {X 0,Y 499.864,Z 439.891,A -85,B 0,C 180,E1 19427.054,E2 19427.054} C_VEL
LIN {X 0,Y 503.717,Z 445.37,A -85,B 0,C 180,E1 19424.692,E2 19424.692} C_VEL
LIN {X 0,Y 506.818,Z 449.71,A -85,B 0,C 180,E1 19423.088,E2 19423.088} C_VEL
LIN {X 0,Y 511.163,Z 456.011,A -85,B 0,C 180,E1 19421.111,E2 19421.111} C_VEL
LIN {X 0,Y 516.013,Z 463.122,A -85,B 0,C 180,E1 19419.171,E2 19419.171} C_VEL
LIN {X 0,Y 523.708,Z 475.097,A -85,B 0,C 180,E1 19416.482,E2 19416.482} C_VEL
LIN {X 0,Y 529.48,Z 484.849,A -85,B 0,C 180,E1 19414.684,E2 19414.684} C_VEL
LIN {X 0,Y 515.021,Z 696.435,A -85,B 0,C 180,E1 19411.333,E2 19411.333} C_VEL
LIN {X 0,Y 506.991,Z 817.099,A -85,B 0,C 180,E1 19409.405,E2 19409.405} C_VEL
LIN {X 0,Y 503.814,Z 845.03,A -85,B 0,C 180,E1 19408.861,E2 19408.861} C_VEL
LIN {X 0,Y 499.727,Z 870.103,A -85,B 0,C 180,E1 19408.222,E2 19408.222} C_VEL
LIN {X 0,Y 495.598,Z 891.407,A -85,B 0,C 180,E1 19407.543,E2 19407.543} C_VEL
LIN {X 0,Y 490.9,Z 912.507,A -85,B 0,C 180,E1 19406.731,E2 19406.731} C_VEL
LIN {X 0,Y 484.663,Z 937.426,A -85,B 0,C 180,E1 19405.578,E2 19405.578} C_VEL
LIN {X 0,Y 477.663,Z 961.711,A -85,B 0,C 180,E1 19404.206,E2 19404.206} C_VEL
LIN {X 0,Y 471.423,Z 981.677,A -85,B 0,C 180,E1 19402.889,E2 19402.889} C_VEL
LIN {X 0,Y 464.989,Z 1001.004,A -85,B 0,C 180,E1 19401.42,E2 19401.42} C_VEL
LIN {X 0,Y 456.917,Z 1023.955,A -85,B 0,C 180,E1 19399.405,E2 19399.405} C_VEL
LIN {X 0,Y 449.015,Z 1044.977,A -85,B 0,C 180,E1 19397.219,E2 19397.219} C_VEL
LIN {X 0,Y 442.337,Z 1062.375,A -85,B 0,C 180,E1 19395.149,E2 19395.149} C_VEL
LIN {X 0,Y 435.591,Z 1079.738,A -85,B 0,C 180,E1 19392.8,E2 19392.8} C_VEL
LIN {X 0,Y 427.814,Z 1099.801,A -85,B 0,C 180,E1 19389.646,E2 19389.646} C_VEL
LIN {X 0,Y 422.183,Z 1114.478,A -85,B 0,C 180,E1 19386.981,E2 19386.981} C_VEL
LIN {X 0,Y 417.526,Z 1127.039,A -85,B 0,C 180,E1 19384.413,E2 19384.413} C_VEL
LIN {X 0,Y 413.131,Z 1139.592,A -85,B 0,C 180,E1 19381.518,E2 19381.518} C_VEL
LIN {X 0,Y 408.55,Z 1153.885,A -85,B 0,C 180,E1 19377.71,E2 19377.71} C_VEL
LIN {X 0,Y 405.608,Z 1164.247,A -85,B 0,C 180,E1 19374.465,E2 19374.465} C_VEL
LIN {X 0,Y 403.495,Z 1172.837,A -85,B 0,C 180,E1 19371.362,E2 19371.362} C_VEL
LIN {X 0,Y 402.043,Z 1179.878,A -85,B 0,C 180,E1 19368.412,E2 19368.412} C_VEL
LIN {X 0,Y 401.06,Z 1186.118,A -85,B 0,C 180,E1 19365.323,E2 19365.323} C_VEL
LIN {X 0,Y 400.421,Z 1191.653,A -85,B 0,C 180,E1 19361.961,E2 19361.961} C_VEL
LIN {X 0,Y 400.137,Z 1196.248,A -85,B 0,C 180,E1 19358.189,E2 19358.189} C_VEL
LIN {X 0,Y 400.091,Z 1198.839,A -85,B 0,C 180,E1 19354.874,E2 19354.874} C_VEL
LIN {X 0,Y 400.094,Z 1200.079,A -85,B 0,C 180,E1 19351.862,E2 19351.862} C_VEL
LIN {X 0,Y 400.093,Z 1200.246,A -85,B 0,C 180,E1 19348.998,E2 19348.998} C_VEL
LIN {X 0,Y 400.081,Z 1199.415,A -85,B 0,C 180,E1 19346.131,E2 19346.131} C_VEL
LIN {X 0,Y 400.094,Z 1197.585,A -85,B 0,C 180,E1 19343.255,E2 19343.255} C_VEL
LIN {X 0,Y 400.208,Z 1194.749,A -85,B 0,C 180,E1 19340.364,E2 19340.364} C_VEL
LIN {X 0,Y 400.495,Z 1190.889,A -85,B 0,C 180,E1 19337.455,E2 19337.455} C_VEL
LIN {X 0,Y 401.097,Z 1185.984,A -85,B 0,C 180,E1 19334.53,E2 19334.53} C_VEL
LIN {X 0,Y 402.045,Z 1179.999,A -85,B 0,C 180,E1 19331.589,E2 19331.589} C_VEL
LIN {X 0,Y 403.499,Z 1172.9,A -85,B 0,C 180,E1 19328.638,E2 19328.638} C_VEL
LIN {X 0,Y 405.724,Z 1163.76,A -85,B 0,C 180,E1 19325.388,E2 19325.388} C_VEL
LIN {X 0,Y 409.328,Z 1150.962,A -85,B 0,C 180,E1 19321.555,E2 19321.555} C_VEL
LIN {X 0,Y 412.886,Z 1139.511,A -85,B 0,C 180,E1 19318.624,E2 19318.624} C_VEL
LIN {X 0,Y 416.945,Z 1127.267,A -85,B 0,C 180,E1 19315.865,E2 19315.865} C_VEL
LIN {X 0,Y 421.463,Z 1114.329,A -85,B 0,C 180,E1 19313.285,E2 19313.285} C_VEL
LIN {X 0,Y 427.614,Z 1097.258,A -85,B 0,C 180,E1 19310.292,E2 19310.292} C_VEL
LIN {X 0,Y 434.092,Z 1078.996,A -85,B 0,C 180,E1 19307.556,E2 19307.556} C_VEL
LIN {X 0,Y 439.945,Z 1062.559,A -85,B 0,C 180,E1 19305.391,E2 19305.391} C_VEL
LIN {X 0,Y 446.142,Z 1044.873,A -85,B 0,C 180,E1 19303.335,E2 19303.335} C_VEL
LIN {X 0,Y 454.114,Z 1021.132,A -85,B 0,C 180,E1 19300.957,E2 19300.957} C_VEL
LIN {X 0,Y 460.379,Z 1001.384,A -85,B 0,C 180,E1 19299.263,E2 19299.263} C_VEL
LIN {X 0,Y 466.008,Z 982.648,A -85,B 0,C 180,E1 19297.855,E2 19297.855} C_VEL
LIN {X 0,Y 471.651,Z 962.614,A -85,B 0,C 180,E1 19296.54,E2 19296.54} C_VEL
LIN {X 0,Y 478.216,Z 936.923,A -85,B 0,C 180,E1 19295.099,E2 19295.099} C_VEL
LIN {X 0,Y 483.408,Z 913.773,A -85,B 0,C 180,E1 19294.027,E2 19294.027} C_VEL
LIN {X 0,Y 487.598,Z 892.846,A -85,B 0,C 180,E1 19293.214,E2 19293.214} C_VEL
LIN {X 0,Y 491.37,Z 871.083,A -85,B 0,C 180,E1 19292.508,E2 19292.508} C_VEL
LIN {X 0,Y 495.29,Z 844.015,A -85,B 0,C 180,E1 19291.815,E2 19291.815} C_VEL
LIN {X 0,Y 497.887,Z 817.372,A -85,B 0,C 180,E1 19291.302,E2 19291.302} C_VEL
LIN {X 0,Y 509.257,Z 612.682,A -85,B 0,C 180,E1 19288.094,E2 19288.094} C_VEL
LIN {X 0,Y 516.748,Z 479.735,A -85,B 0,C 180,E1 19285.994,E2 19285.994} C_VEL
LIN {X 0,Y 505.14,Z 461.023,A -85,B 0,C 180,E1 19283.291,E2 19283.291} C_VEL
LIN {X 0,Y 494.369,Z 444.611,A -85,B 0,C 180,E1 19280.481,E2 19280.481} C_VEL
LIN {X 0,Y 485.829,Z 432.272,A -85,B 0,C 180,E1 19277.982,E2 19277.982} C_VEL
LIN {X 0,Y 478.913,Z 422.623,A -85,B 0,C 180,E1 19275.718,E2 19275.718} C_VEL
LIN {X 0,Y 471.869,Z 413.179,A -85,B 0,C 180,E1 19273.105,E2 19273.105} C_VEL
LIN {X 0,Y 467.781,Z 407.883,A -85,B 0,C 180,E1 19271.404,E2 19271.404} C_VEL
LIN {X 0,Y 463.433,Z 402.251,A -85,B 0,C 180,E1 19269.375,E2 19269.375} C_VEL
LIN {X 0,Y 459.464,Z 397.291,A -85,B 0,C 180,E1 19267.251,E2 19267.251} C_VEL
LIN {X 0,Y 455.399,Z 392.207,A -85,B 0,C 180,E1 19264.66,E2 19264.66} C_VEL
LIN {X 0,Y 450.695,Z 386.406,A -85,B 0,C 180,E1 19260.636,E2 19260.636} C_VEL
LIN {X 0,Y 447.325,Z 382.939,A -85,B 0,C 180,E1 19254.87,E2 19254.87} C_VEL
LIN {X 0,Y 447.172,Z 382.706,A -85,B 0,C 180,E1 19251.772,E2 19251.772} C_VEL
LIN {X 0,Y 448.664,Z 384.64,A -85,B 0,C 180,E1 19247.516,E2 19247.516} C_VEL
LIN {X 0,Y 451.164,Z 386.922,A -85,B 0,C 180,E1 19244.445,E2 19244.445} C_VEL
LIN {X 0,Y 454.85,Z 391.693,A -85,B 0,C 180,E1 19241.28,E2 19241.28} C_VEL
LIN {X 0,Y 456.302,Z 393.361,A -85,B 0,C 180,E1 19240.278,E2 19240.278} C_VEL
LIN {X 0,Y 460.854,Z 399.072,A -85,B 0,C 180,E1 19237.551,E2 19237.551} C_VEL
LIN {X 0,Y 464.955,Z 404.228,A -85,B 0,C 180,E1 19235.477,E2 19235.477} C_VEL
LIN {X 0,Y 469.384,Z 410.015,A -85,B 0,C 180,E1 19233.495,E2 19233.495} C_VEL
LIN {X 0,Y 473.73,Z 415.775,A -85,B 0,C 180,E1 19231.75,E2 19231.75} C_VEL
LIN {X 0,Y 479.781,Z 423.989,A -85,B 0,C 180,E1 19229.574,E2 19229.574} C_VEL
LIN {X 0,Y 487.685,Z 435.178,A -85,B 0,C 180,E1 19227.055,E2 19227.055} C_VEL
LIN {X 0,Y 496.198,Z 447.773,A -85,B 0,C 180,E1 19224.631,E2 19224.631} C_VEL
LIN {X 0,Y 505.8,Z 462.716,A -85,B 0,C 180,E1 19222.17,E2 19222.17} C_VEL
LIN {X 0,Y 512.371,Z 473.684,A -85,B 0,C 180,E1 19220.611,E2 19220.611} C_VEL
LIN {X 0,Y 498.966,Z 705.016,A -85,B 0,C 180,E1 19217.061,E2 19217.061} C_VEL
LIN {X 0,Y 493.907,Z 791.984,A -85,B 0,C 180,E1 19215.702,E2 19215.702} C_VEL
LIN {X 0,Y 491.073,Z 819.77,A -85,B 0,C 180,E1 19215.117,E2 19215.117} C_VEL
LIN {X 0,Y 487.879,Z 842.661,A -85,B 0,C 180,E1 19214.463,E2 19214.463} C_VEL
LIN {X 0,Y 484.632,Z 861.9,A -85,B 0,C 180,E1 19213.789,E2 19213.789} C_VEL
LIN {X 0,Y 480.376,Z 883.497,A -85,B 0,C 180,E1 19212.888,E2 19212.888} C_VEL
LIN {X 0,Y 474.491,Z 908.962,A -85,B 0,C 180,E1 19211.588,E2 19211.588} C_VEL
LIN {X 0,Y 469.466,Z 928.077,A -85,B 0,C 180,E1 19210.43,E2 19210.43} C_VEL
LIN {X 0,Y 463.938,Z 947.35,A -85,B 0,C 180,E1 19209.078,E2 19209.078} C_VEL
LIN {X 0,Y 456.914,Z 969.811,A -85,B 0,C 180,E1 19207.233,E2 19207.233} C_VEL
LIN {X 0,Y 450.46,Z 988.714,A -85,B 0,C 180,E1 19205.403,E2 19205.403} C_VEL
LIN {X 0,Y 444.407,Z 1005.605,A -85,B 0,C 180,E1 19203.528,E2 19203.528} C_VEL
LIN {X 0,Y 437.38,Z 1024.445,A -85,B 0,C 180,E1 19201.107,E2 19201.107} C_VEL
LIN {X 0,Y 431.118,Z 1040.467,A -85,B 0,C 180,E1 19198.69,E2 19198.69} C_VEL
LIN {X 0,Y 425.774,Z 1054.048,A -85,B 0,C 180,E1 19196.349,E2 19196.349} C_VEL
LIN {X 0,Y 420.009,Z 1068.806,A -85,B 0,C 180,E1 19193.425,E2 19193.425} C_VEL
LIN {X 0,Y 414.863,Z 1082.012,A -85,B 0,C 180,E1 19190.307,E2 19190.307} C_VEL
LIN {X 0,Y 410.947,Z 1092.596,A -85,B 0,C 180,E1 19187.413,E2 19187.413} C_VEL
LIN {X 0,Y 407.113,Z 1103.806,A -85,B 0,C 180,E1 19183.782,E2 19183.782} C_VEL
LIN {X 0,Y 404.553,Z 1112.041,A -85,B 0,C 180,E1 19180.538,E2 19180.538} C_VEL
LIN {X 0,Y 402.955,Z 1118.038,A -85,B 0,C 180,E1 19177.734,E2 19177.734} C_VEL
LIN {X 0,Y 401.505,Z 1120.25,A -85,B 0,C 180,E1 19176.691,E2 19176.691} C_VEL
LIN {X 0,Y 394.16,Z 1125.694,A -85,B 0,C 180,E1 19173.834,E2 19173.834} C_VEL
LIN {X 0,Y 393.3,Z 1126.882,A -85,B 0,C 180,E1 19172.971,E2 19172.971} C_VEL
LIN {X 0,Y 392.721,Z 1130.485,A -85,B 0,C 180,E1 19169.854,E2 19169.854} C_VEL
LIN {X 0,Y 392.422,Z 1133.341,A -85,B 0,C 180,E1 19166.348,E2 19166.348} C_VEL
LIN {X 0,Y 392.319,Z 1134.809,A -85,B 0,C 180,E1 19162.679,E2 19162.679} C_VEL
LIN {X 0,Y 392.317,Z 1134.983,A -85,B 0,C 180,E1 19159.575,E2 19159.575} C_VEL
LIN {X 0,Y 392.405,Z 1134.221,A -85,B 0,C 180,E1 19156.593,E2 19156.593} C_VEL
LIN {X 0,Y 392.618,Z 1132.526,A -85,B 0,C 180,E1 19153.58,E2 19153.58} C_VEL
LIN {X 0,Y 393.205,Z 1129.276,A -85,B 0,C 180,E1 19149.923,E2 19149.923} C_VEL
LIN {X 0,Y 394.39,Z 1124.146,A -85,B 0,C 180,E1 19146.069,E2 19146.069} C_VEL
LIN {X 0,Y 395.929,Z 1118.873,A -85,B 0,C 180,E1 19142.963,E2 19142.963} C_VEL
LIN {X 0,Y 398.261,Z 1112.124,A -85,B 0,C 180,E1 19139.694,E2 19139.694} C_VEL
LIN {X 0,Y 402.105,Z 1102.258,A -85,B 0,C 180,E1 19135.808,E2 19135.808} C_VEL
LIN {X 0,Y 406.109,Z 1092.823,A -85,B 0,C 180,E1 19132.723,E2 19132.723} C_VEL
LIN {X 0,Y 411.017,Z 1081.971,A -85,B 0,C 180,E1 19129.678,E2 19129.678} C_VEL
LIN {X 0,Y 417.772,Z 1067.409,A -85,B 0,C 180,E1 19126.238,E2 19126.238} C_VEL
LIN {X 0,Y 423.924,Z 1054.289,A -85,B 0,C 180,E1 19123.607,E2 19123.607} C_VEL
LIN {X 0,Y 430.839,Z 1039.533,A -85,B 0,C 180,E1 19121.041,E2 19121.041} C_VEL
LIN {X 0,Y 439.162,Z 1021.196,A -85,B 0,C 180,E1 19118.34,E2 19118.34} C_VEL
LIN {X 0,Y 445.891,Z 1005.776,A -85,B 0,C 180,E1 19116.388,E2 19116.388} C_VEL
LIN {X 0,Y 452.829,Z 989.196,A -85,B 0,C 180,E1 19114.554,E2 19114.554} C_VEL
LIN {X 0,Y 461.291,Z 967.689,A -85,B 0,C 180,E1 19112.518,E2 19112.518} C_VEL
LIN {X 0,Y 468.182,Z 948.467,A -85,B 0,C 180,E1 19110.978,E2 19110.978} C_VEL
LIN {X 0,Y 474.288,Z 930.029,A -85,B 0,C 180,E1 19109.698,E2 19109.698} C_VEL
LIN {X 0,Y 480.835,Z 908.334,A -85,B 0,C 180,E1 19108.407,E2 19108.407} C_VEL
LIN {X 0,Y 487.291,Z 883.536,A -85,B 0,C 180,E1 19107.191,E2 19107.191} C_VEL
LIN {X 0,Y 492.021,Z 862.474,A -85,B 0,C 180,E1 19106.34,E2 19106.34} C_VEL
LIN {X 0,Y 495.97,Z 841.891,A -85,B 0,C 180,E1 19105.651,E2 19105.651} C_VEL
LIN {X 0,Y 499.985,Z 815.837,A -85,B 0,C 180,E1 19104.957,E2 19104.957} C_VEL
LIN {X 0,Y 502.583,Z 791.91,A -85,B 0,C 180,E1 19104.484,E2 19104.484} C_VEL
LIN {X 0,Y 518.654,Z 562.795,A -85,B 0,C 180,E1 19100.935,E2 19100.935} C_VEL
LIN {X 0,Y 524.143,Z 486.404,A -85,B 0,C 180,E1 19099.752,E2 19099.752} C_VEL
LIN {X 0,Y 516.199,Z 473.61,A -85,B 0,C 180,E1 19097.036,E2 19097.036} C_VEL
LIN {X 0,Y 510.42,Z 464.782,A -85,B 0,C 180,E1 19094.754,E2 19094.754} C_VEL
LIN {X 0,Y 505.949,Z 458.302,A -85,B 0,C 180,E1 19092.73,E2 19092.73} C_VEL
LIN {X 0,Y 503.16,Z 454.2,A -85,B 0,C 180,E1 19091.288,E2 19091.288} C_VEL
LIN {X 0,Y 500.175,Z 449.974,A -85,B 0,C 180,E1 19089.551,E2 19089.551} C_VEL
LIN {X 0,Y 497.542,Z 446.16,A -85,B 0,C 180,E1 19087.738,E2 19087.738} C_VEL
LIN {X 0,Y 494.097,Z 441.227,A -85,B 0,C 180,E1 19084.643,E2 19084.643} C_VEL
LIN {X 0,Y 491.123,Z 437.367,A -85,B 0,C 180,E1 19079.183,E2 19079.183} C_VEL
LIN {X 0,Y 491.121,Z 437.342,A -85,B 0,C 180,E1 19076.615,E2 19076.615} C_VEL
LIN {X 0,Y 493.228,Z 440.47,A -85,B 0,C 180,E1 19072.076,E2 19072.076} C_VEL
LIN {X 0,Y 494.744,Z 442.161,A -85,B 0,C 180,E1 19070.402,E2 19070.402} C_VEL
LIN {X 0,Y 498.55,Z 447.586,A -85,B 0,C 180,E1 19067.255,E2 19067.255} C_VEL
LIN {X 0,Y 502.225,Z 452.92,A -85,B 0,C 180,E1 19064.941,E2 19064.941} C_VEL
LIN {X 0,Y 505.382,Z 457.461,A -85,B 0,C 180,E1 19063.269,E2 19063.269} C_VEL
LIN {X 0,Y 509.652,Z 463.753,A -85,B 0,C 180,E1 19061.29,E2 19061.29} C_VEL
LIN {X 0,Y 514.509,Z 471.056,A -85,B 0,C 180,E1 19059.316,E2 19059.316} C_VEL
LIN {X 0,Y 521.652,Z 482.386,A -85,B 0,C 180,E1 19056.773,E2 19056.773} C_VEL
LIN {X 0,Y 525.884,Z 489.785,A -85,B 0,C 180,E1 19055.404,E2 19055.404} C_VEL
LIN {X 0,Y 510.921,Z 702.664,A -85,B 0,C 180,E1 19052.032,E2 19052.032} C_VEL
LIN {X 0,Y 503.076,Z 816.898,A -85,B 0,C 180,E1 19050.203,E2 19050.203} C_VEL
LIN {X 0,Y 499.786,Z 844.995,A -85,B 0,C 180,E1 19049.655,E2 19049.655} C_VEL
LIN {X 0,Y 495.65,Z 869.744,A -85,B 0,C 180,E1 19049.027,E2 19049.027} C_VEL
LIN {X 0,Y 491.448,Z 890.866,A -85,B 0,C 180,E1 19048.358,E2 19048.358} C_VEL
LIN {X 0,Y 486.808,Z 911.204,A -85,B 0,C 180,E1 19047.582,E2 19047.582} C_VEL
LIN {X 0,Y 481.061,Z 933.625,A -85,B 0,C 180,E1 19046.563,E2 19046.563} C_VEL
LIN {X 0,Y 473.412,Z 959.923,A -85,B 0,C 180,E1 19045.113,E2 19045.113} C_VEL
LIN {X 0,Y 466.758,Z 980.633,A -85,B 0,C 180,E1 19043.754,E2 19043.754} C_VEL
LIN {X 0,Y 460.366,Z 999.317,A -85,B 0,C 180,E1 19042.34,E2 19042.34} C_VEL
LIN {X 0,Y 453.503,Z 1018.256,A -85,B 0,C 180,E1 19040.702,E2 19040.702} C_VEL
LIN {X 0,Y 444.685,Z 1041.307,A -85,B 0,C 180,E1 19038.384,E2 19038.384} C_VEL
LIN {X 0,Y 437.219,Z 1060.009,A -85,B 0,C 180,E1 19036.179,E2 19036.179} C_VEL
LIN {X 0,Y 430.565,Z 1076.419,A -85,B 0,C 180,E1 19033.974,E2 19033.974} C_VEL
LIN {X 0,Y 423.294,Z 1094.376,A -85,B 0,C 180,E1 19031.225,E2 19031.225} C_VEL
LIN {X 0,Y 416.288,Z 1111.75,A -85,B 0,C 180,E1 19028.117,E2 19028.117} C_VEL
LIN {X 0,Y 411.065,Z 1125.141,A -85,B 0,C 180,E1 19025.373,E2 19025.373} C_VEL
LIN {X 0,Y 406.558,Z 1137.194,A -85,B 0,C 180,E1 19022.588,E2 19022.588} C_VEL
LIN {X 0,Y 402.441,Z 1149.09,A -85,B 0,C 180,E1 19019.467,E2 19019.467} C_VEL
LIN {X 0,Y 398.272,Z 1162.544,A -85,B 0,C 180,E1 19015.336,E2 19015.336} C_VEL
LIN {X 0,Y 395.876,Z 1171.608,A -85,B 0,C 180,E1 19012.034,E2 19012.034} C_VEL
LIN {X 0,Y 394.244,Z 1178.96,A -85,B 0,C 180,E1 19008.912,E2 19008.912} C_VEL
LIN {X 0,Y 393.179,Z 1185.181,A -85,B 0,C 180,E1 19005.789,E2 19005.789} C_VEL
LIN {X 0,Y 392.518,Z 1190.316,A -85,B 0,C 180,E1 19002.654,E2 19002.654} C_VEL
LIN {X 0,Y 392.187,Z 1194.846,A -85,B 0,C 180,E1 18999.095,E2 18999.095} C_VEL
LIN {X 0,Y 392.109,Z 1197.948,A -85,B 0,C 180,E1 18995.414,E2 18995.414} C_VEL
LIN {X 0,Y 392.12,Z 1199.394,A -85,B 0,C 180,E1 18992.046,E2 18992.046} C_VEL
LIN {X 0,Y 392.116,Z 1199.61,A -85,B 0,C 180,E1 18989.123,E2 18989.123} C_VEL
LIN {X 0,Y 392.105,Z 1198.825,A -85,B 0,C 180,E1 18986.199,E2 18986.199} C_VEL
LIN {X 0,Y 392.116,Z 1196.913,A -85,B 0,C 180,E1 18983.117,E2 18983.117} C_VEL
LIN {X 0,Y 392.236,Z 1194.062,A -85,B 0,C 180,E1 18980.166,E2 18980.166} C_VEL
LIN {X 0,Y 392.536,Z 1190.184,A -85,B 0,C 180,E1 18977.197,E2 18977.197} C_VEL
LIN {X 0,Y 393.178,Z 1185.256,A -85,B 0,C 180,E1 18974.211,E2 18974.211} C_VEL
LIN {X 0,Y 394.191,Z 1179.243,A -85,B 0,C 180,E1 18971.208,E2 18971.208} C_VEL
LIN {X 0,Y 395.733,Z 1172.113,A -85,B 0,C 180,E1 18968.198,E2 18968.198} C_VEL
LIN {X 0,Y 398.081,Z 1162.934,A -85,B 0,C 180,E1 18964.883,E2 18964.883} C_VEL
LIN {X 0,Y 401.895,Z 1150.075,A -85,B 0,C 180,E1 18960.979,E2 18960.979} C_VEL
LIN {X 0,Y 405.623,Z 1138.564,A -85,B 0,C 180,E1 18957.994,E2 18957.994} C_VEL
LIN {X 0,Y 409.653,Z 1126.972,A -85,B 0,C 180,E1 18955.341,E2 18955.341} C_VEL
LIN {X 0,Y 414.626,Z 1113.299,A -85,B 0,C 180,E1 18952.577,E2 18952.577} C_VEL
LIN {X 0,Y 421.299,Z 1095.342,A -85,B 0,C 180,E1 18949.418,E2 18949.418} C_VEL
LIN {X 0,Y 427.779,Z 1077.802,A -85,B 0,C 180,E1 18946.777,E2 18946.777} C_VEL
LIN {X 0,Y 433.547,Z 1062.171,A -85,B 0,C 180,E1 18944.702,E2 18944.702} C_VEL
LIN {X 0,Y 439.921,Z 1044.548,A -85,B 0,C 180,E1 18942.635,E2 18942.635} C_VEL
LIN {X 0,Y 447.833,Z 1021.836,A -85,B 0,C 180,E1 18940.329,E2 18940.329} C_VEL
LIN {X 0,Y 454.53,Z 1001.337,A -85,B 0,C 180,E1 18938.555,E2 18938.555} C_VEL
LIN {X 0,Y 460.565,Z 981.781,A -85,B 0,C 180,E1 18937.078,E2 18937.078} C_VEL
LIN {X 0,Y 466.635,Z 960.765,A -85,B 0,C 180,E1 18935.7,E2 18935.7} C_VEL
LIN {X 0,Y 473.496,Z 934.271,A -85,B 0,C 180,E1 18934.238,E2 18934.238} C_VEL
LIN {X 0,Y 478.496,Z 912.45,A -85,B 0,C 180,E1 18933.237,E2 18933.237} C_VEL
LIN {X 0,Y 482.655,Z 892.092,A -85,B 0,C 180,E1 18932.45,E2 18932.45} C_VEL
LIN {X 0,Y 486.705,Z 869.232,A -85,B 0,C 180,E1 18931.715,E2 18931.715} C_VEL
LIN {X 0,Y 490.866,Z 840.018,A -85,B 0,C 180,E1 18930.993,E2 18930.993} C_VEL
LIN {X 0,Y 493.183,Z 816.08,A -85,B 0,C 180,E1 18930.536,E2 18930.536} C_VEL
LIN {X 0,Y 505.181,Z 606.433,A -85,B 0,C 180,E1 18927.241,E2 18927.241} C_VEL
LIN {X 0,Y 512.311,Z 483.992,A -85,B 0,C 180,E1 18925.305,E2 18925.305} C_VEL
LIN {X 0,Y 501.053,Z 465.754,A -85,B 0,C 180,E1 18922.591,E2 18922.591} C_VEL
LIN {X 0,Y 490.922,Z 450.138,A -85,B 0,C 180,E1 18919.854,E2 18919.854} C_VEL
LIN {X 0,Y 480.881,Z 435.417,A -85,B 0,C 180,E1 18916.768,E2 18916.768} C_VEL
LIN {X 0,Y 472.824,Z 424.403,A -85,B 0,C 180,E1 18913.913,E2 18913.913} C_VEL
LIN {X 0,Y 469.532,Z 419.977,A -85,B 0,C 180,E1 18912.608,E2 18912.608} C_VEL
LIN {X 0,Y 466.088,Z 415.39,A -85,B 0,C 180,E1 18911.132,E2 18911.132} C_VEL
LIN {X 0,Y 461.818,Z 409.772,A -85,B 0,C 180,E1 18909.094,E2 18909.094} C_VEL
LIN {X 0,Y 458.138,Z 405.065,A -85,B 0,C 180,E1 18907.083,E2 18907.083} C_VEL
LIN {X 0,Y 454.044,Z 399.912,A -85,B 0,C 180,E1 18904.421,E2 18904.421} C_VEL
LIN {X 0,Y 449.591,Z 394.277,A -85,B 0,C 180,E1 18900.51,E2 18900.51} C_VEL
LIN {X 0,Y 446.323,Z 390.837,A -85,B 0,C 180,E1 18894.73,E2 18894.73} C_VEL
LIN {X 0,Y 446.212,Z 390.667,A -85,B 0,C 180,E1 18891.625,E2 18891.625} C_VEL
LIN {X 0,Y 447.87,Z 392.78,A -85,B 0,C 180,E1 18887.231,E2 18887.231} C_VEL
LIN {X 0,Y 450.084,Z 394.843,A -85,B 0,C 180,E1 18884.539,E2 18884.539} C_VEL
LIN {X 0,Y 453.741,Z 399.601,A -85,B 0,C 180,E1 18881.359,E2 18881.359} C_VEL
LIN {X 0,Y 455.251,Z 401.499,A -85,B 0,C 180,E1 18880.297,E2 18880.297} C_VEL
LIN {X 0,Y 459.456,Z 406.805,A -85,B 0,C 180,E1 18877.749,E2 18877.749} C_VEL
LIN {X 0,Y 463.373,Z 411.814,A -85,B 0,C 180,E1 18875.728,E2 18875.728} C_VEL
LIN {X 0,Y 467.675,Z 417.517,A -85,B 0,C 180,E1 18873.766,E2 18873.766} C_VEL
LIN {X 0,Y 472.034,Z 423.394,A -85,B 0,C 180,E1 18871.983,E2 18871.983} C_VEL
LIN {X 0,Y 477.841,Z 431.421,A -85,B 0,C 180,E1 18869.854,E2 18869.854} C_VEL
LIN {X 0,Y 486.197,Z 443.417,A -85,B 0,C 180,E1 18867.152,E2 18867.152} C_VEL
LIN {X 0,Y 495.055,Z 456.843,A -85,B 0,C 180,E1 18864.608,E2 18864.608} C_VEL
LIN {X 0,Y 504.851,Z 472.468,A -85,B 0,C 180,E1 18862.086,E2 18862.086} C_VEL
LIN {X 0,Y 507.999,Z 478.005,A -85,B 0,C 180,E1 18861.32,E2 18861.32} C_VEL
LIN {X 0,Y 494.187,Z 709.604,A -85,B 0,C 180,E1 18857.755,E2 18857.755} C_VEL
LIN {X 0,Y 489.221,Z 792.307,A -85,B 0,C 180,E1 18856.457,E2 18856.457} C_VEL
LIN {X 0,Y 486.34,Z 819.975,A -85,B 0,C 180,E1 18855.875,E2 18855.875} C_VEL
LIN {X 0,Y 483.066,Z 842.907,A -85,B 0,C 180,E1 18855.22,E2 18855.22} C_VEL
LIN {X 0,Y 479.846,Z 861.577,A -85,B 0,C 180,E1 18854.57,E2 18854.57} C_VEL
LIN {X 0,Y 475.524,Z 883.067,A -85,B 0,C 180,E1 18853.679,E2 18853.679} C_VEL
LIN {X 0,Y 469.5,Z 908.687,A -85,B 0,C 180,E1 18852.378,E2 18852.378} C_VEL
LIN {X 0,Y 464.095,Z 928.738,A -85,B 0,C 180,E1 18851.161,E2 18851.161} C_VEL
LIN {X 0,Y 458.415,Z 947.998,A -85,B 0,C 180,E1 18849.803,E2 18849.803} C_VEL
LIN {X 0,Y 450.964,Z 971.088,A -85,B 0,C 180,E1 18847.89,E2 18847.89} C_VEL
LIN {X 0,Y 444.54,Z 989.367,A -85,B 0,C 180,E1 18846.106,E2 18846.106} C_VEL
LIN {X 0,Y 438.296,Z 1006.253,A -85,B 0,C 180,E1 18844.217,E2 18844.217} C_VEL
LIN {X 0,Y 430.672,Z 1025.96,A -85,B 0,C 180,E1 18841.647,E2 18841.647} C_VEL
LIN {X 0,Y 424.551,Z 1041.124,A -85,B 0,C 180,E1 18839.331,E2 18839.331} C_VEL
LIN {X 0,Y 419.009,Z 1054.701,A -85,B 0,C 180,E1 18836.961,E2 18836.961} C_VEL
LIN {X 0,Y 413.018,Z 1069.456,A -85,B 0,C 180,E1 18833.998,E2 18833.998} C_VEL
LIN {X 0,Y 407.649,Z 1082.672,A -85,B 0,C 180,E1 18830.833,E2 18830.833} C_VEL
LIN {X 0,Y 403.561,Z 1093.252,A -85,B 0,C 180,E1 18827.892,E2 18827.892} C_VEL
LIN {X 0,Y 399.538,Z 1104.463,A -85,B 0,C 180,E1 18824.196,E2 18824.196} C_VEL
LIN {X 0,Y 396.843,Z 1112.7,A -85,B 0,C 180,E1 18820.892,E2 18820.892} C_VEL
LIN {X 0,Y 394.995,Z 1119.321,A -85,B 0,C 180,E1 18817.71,E2 18817.71} C_VEL
LIN {X 0,Y 393.523,Z 1125.807,A -85,B 0,C 180,E1 18813.788,E2 18813.788} C_VEL
LIN {X 0,Y 393.3,Z 1126.882,A -85,B 0,C 180,E1 18812.971,E2 18812.971} C_VEL
LIN {X 0,Y 392.078,Z 1128.457,A -85,B 0,C 180,E1 18811.874,E2 18811.874} C_VEL
LIN {X 0,Y 385.183,Z 1132.253,A -85,B 0,C 180,E1 18808.781,E2 18808.781} C_VEL
LIN {X 0,Y 384.56,Z 1132.882,A -85,B 0,C 180,E1 18807.962,E2 18807.962} C_VEL
LIN {X 0,Y 384.381,Z 1134.695,A -85,B 0,C 180,E1 18804.926,E2 18804.926} C_VEL
LIN {X 0,Y 384.351,Z 1135.58,A -85,B 0,C 180,E1 18801.924,E2 18801.924} C_VEL
LIN {X 0,Y 384.359,Z 1135.553,A -85,B 0,C 180,E1 18798.74,E2 18798.74} C_VEL
LIN {X 0,Y 384.534,Z 1134.346,A -85,B 0,C 180,E1 18795.083,E2 18795.083} C_VEL
LIN {X 0,Y 384.966,Z 1131.592,A -85,B 0,C 180,E1 18791.369,E2 18791.369} C_VEL
LIN {X 0,Y 385.704,Z 1128.132,A -85,B 0,C 180,E1 18788.137,E2 18788.137} C_VEL
LIN {X 0,Y 386.955,Z 1123.647,A -85,B 0,C 180,E1 18784.928,E2 18784.928} C_VEL
LIN {X 0,Y 389.341,Z 1116.61,A -85,B 0,C 180,E1 18780.963,E2 18780.963} C_VEL
LIN {X 0,Y 392.37,Z 1108.755,A -85,B 0,C 180,E1 18777.474,E2 18777.474} C_VEL
LIN {X 0,Y 395.979,Z 1100.329,A -85,B 0,C 180,E1 18774.318,E2 18774.318} C_VEL
LIN {X 0,Y 401.25,Z 1089.002,A -85,B 0,C 180,E1 18770.733,E2 18770.733} C_VEL
LIN {X 0,Y 407.214,Z 1076.442,A -85,B 0,C 180,E1 18767.446,E2 18767.446} C_VEL
LIN {X 0,Y 412.97,Z 1064.692,A -85,B 0,C 180,E1 18764.795,E2 18764.795} C_VEL
LIN {X 0,Y 420.368,Z 1049.756,A -85,B 0,C 180,E1 18761.885,E2 18761.885} C_VEL
LIN {X 0,Y 428.238,Z 1033.202,A -85,B 0,C 180,E1 18759.18,E2 18759.18} C_VEL
LIN {X 0,Y 435.297,Z 1018.07,A -85,B 0,C 180,E1 18757.042,E2 18757.042} C_VEL
LIN {X 0,Y 443.707,Z 999.395,A -85,B 0,C 180,E1 18754.76,E2 18754.76} C_VEL
LIN {X 0,Y 452.065,Z 979.22,A -85,B 0,C 180,E1 18752.693,E2 18752.693} C_VEL
LIN {X 0,Y 459.018,Z 961.418,A -85,B 0,C 180,E1 18751.124,E2 18751.124} C_VEL
LIN {X 0,Y 466.859,Z 939.804,A -85,B 0,C 180,E1 18749.485,E2 18749.485} C_VEL
LIN {X 0,Y 474.083,Z 917.112,A -85,B 0,C 180,E1 18748.056,E2 18748.056} C_VEL
LIN {X 0,Y 479.568,Z 898.037,A -85,B 0,C 180,E1 18747.035,E2 18747.035} C_VEL
LIN {X 0,Y 484.686,Z 877.952,A -85,B 0,C 180,E1 18746.113,E2 18746.113} C_VEL
LIN {X 0,Y 490.442,Z 851.308,A -85,B 0,C 180,E1 18745.115,E2 18745.115} C_VEL
LIN {X 0,Y 494.382,Z 828.352,A -85,B 0,C 180,E1 18744.437,E2 18744.437} C_VEL
LIN {X 0,Y 497.436,Z 806.154,A -85,B 0,C 180,E1 18743.93,E2 18743.93} C_VEL
LIN {X 0,Y 500.224,Z 775.72,A -85,B 0,C 180,E1 18743.402,E2 18743.402} C_VEL
LIN {X 0,Y 517.28,Z 537.857,A -85,B 0,C 180,E1 18739.736,E2 18739.736} C_VEL
LIN {X 0,Y 520.737,Z 491.494,A -85,B 0,C 180,E1 18739.023,E2 18739.023} C_VEL
LIN {X 0,Y 513.421,Z 479.47,A -85,B 0,C 180,E1 18736.403,E2 18736.403} C_VEL
LIN {X 0,Y 507.777,Z 470.908,A -85,B 0,C 180,E1 18734.075,E2 18734.075} C_VEL
LIN {X 0,Y 504.172,Z 465.503,A -85,B 0,C 180,E1 18732.368,E2 18732.368} C_VEL
LIN {X 0,Y 501.557,Z 461.603,A -85,B 0,C 180,E1 18730.975,E2 18730.975} C_VEL
LIN {X 0,Y 498.653,Z 457.412,A -85,B 0,C 180,E1 18729.231,E2 18729.231} C_VEL
LIN {X 0,Y 496.252,Z 453.875,A -85,B 0,C 180,E1 18727.526,E2 18727.526} C_VEL
LIN {X 0,Y 493.005,Z 449.105,A -85,B 0,C 180,E1 18724.537,E2 18724.537} C_VEL
LIN {X 0,Y 490.144,Z 445.314,A -85,B 0,C 180,E1 18719.182,E2 18719.182} C_VEL
LIN {X 0,Y 490.143,Z 445.291,A -85,B 0,C 180,E1 18716.608,E2 18716.608} C_VEL
LIN {X 0,Y 492.534,Z 448.728,A -85,B 0,C 180,E1 18711.713,E2 18711.713} C_VEL
LIN {X 0,Y 493.64,Z 450.078,A -85,B 0,C 180,E1 18710.498,E2 18710.498} C_VEL
LIN {X 0,Y 497.321,Z 455.41,A -85,B 0,C 180,E1 18707.4,E2 18707.4} C_VEL
LIN {X 0,Y 500.94,Z 460.775,A -85,B 0,C 180,E1 18705.079,E2 18705.079} C_VEL
LIN {X 0,Y 503.943,Z 465.19,A -85,B 0,C 180,E1 18703.458,E2 18703.458} C_VEL
LIN {X 0,Y 508.151,Z 471.491,A -85,B 0,C 180,E1 18701.471,E2 18701.471} C_VEL
LIN {X 0,Y 513.995,Z 480.458,A -85,B 0,C 180,E1 18699.086,E2 18699.086} C_VEL
LIN {X 0,Y 521.407,Z 492.746,A -85,B 0,C 180,E1 18696.462,E2 18696.462} C_VEL
LIN {X 0,Y 522.376,Z 494.669,A -85,B 0,C 180,E1 18696.136,E2 18696.136} C_VEL
LIN {X 0,Y 506.855,Z 709.64,A -85,B 0,C 180,E1 18692.73,E2 18692.73} C_VEL
LIN {X 0,Y 499.281,Z 816.517,A -85,B 0,C 180,E1 18691.017,E2 18691.017} C_VEL
LIN {X 0,Y 495.899,Z 844.701,A -85,B 0,C 180,E1 18690.467,E2 18690.467} C_VEL
LIN {X 0,Y 491.689,Z 869.327,A -85,B 0,C 180,E1 18689.848,E2 18689.848} C_VEL
LIN {X 0,Y 487.403,Z 890.373,A -85,B 0,C 180,E1 18689.186,E2 18689.186} C_VEL
LIN {X 0,Y 482.389,Z 911.776,A -85,B 0,C 180,E1 18688.371,E2 18688.371} C_VEL
LIN {X 0,Y 475.724,Z 936.928,A -85,B 0,C 180,E1 18687.215,E2 18687.215} C_VEL
LIN {X 0,Y 468.542,Z 960.46,A -85,B 0,C 180,E1 18685.892,E2 18685.892} C_VEL
LIN {X 0,Y 461.983,Z 980.294,A -85,B 0,C 180,E1 18684.588,E2 18684.588} C_VEL
LIN {X 0,Y 455.376,Z 998.992,A -85,B 0,C 180,E1 18683.17,E2 18683.17} C_VEL
LIN {X 0,Y 448.044,Z 1018.563,A -85,B 0,C 180,E1 18681.471,E2 18681.471} C_VEL
LIN {X 0,Y 438.684,Z 1042.07,A -85,B 0,C 180,E1 18679.075,E2 18679.075} C_VEL
LIN {X 0,Y 431.429,Z 1059.601,A -85,B 0,C 180,E1 18676.986,E2 18676.986} C_VEL
LIN {X 0,Y 424.722,Z 1075.504,A -85,B 0,C 180,E1 18674.835,E2 18674.835} C_VEL
LIN {X 0,Y 417.664,Z 1092.156,A -85,B 0,C 180,E1 18672.275,E2 18672.275} C_VEL
LIN {X 0,Y 409.616,Z 1111.224,A -85,B 0,C 180,E1 18668.853,E2 18668.853} C_VEL
LIN {X 0,Y 403.889,Z 1125.26,A -85,B 0,C 180,E1 18665.924,E2 18665.924} C_VEL
LIN {X 0,Y 398.887,Z 1138.054,A -85,B 0,C 180,E1 18662.886,E2 18662.886} C_VEL
LIN {X 0,Y 393.838,Z 1152.173,A -85,B 0,C 180,E1 18659.006,E2 18659.006} C_VEL
LIN {X 0,Y 390.352,Z 1162.985,A -85,B 0,C 180,E1 18655.488,E2 18655.488} C_VEL
LIN {X 0,Y 388.02,Z 1171.424,A -85,B 0,C 180,E1 18652.314,E2 18652.314} C_VEL
LIN {X 0,Y 386.333,Z 1178.669,A -85,B 0,C 180,E1 18649.147,E2 18649.147} C_VEL
LIN {X 0,Y 385.182,Z 1185.084,A -85,B 0,C 180,E1 18645.817,E2 18645.817} C_VEL
LIN {X 0,Y 384.416,Z 1191.206,A -85,B 0,C 180,E1 18641.858,E2 18641.858} C_VEL
LIN {X 0,Y 384.169,Z 1195.309,A -85,B 0,C 180,E1 18638.079,E2 18638.079} C_VEL
LIN {X 0,Y 384.136,Z 1197.601,A -85,B 0,C 180,E1 18634.928,E2 18634.928} C_VEL
LIN {X 0,Y 384.147,Z 1198.765,A -85,B 0,C 180,E1 18631.939,E2 18631.939} C_VEL
LIN {X 0,Y 384.148,Z 1198.927,A -85,B 0,C 180,E1 18628.956,E2 18628.956} C_VEL
LIN {X 0,Y 384.129,Z 1198.085,A -85,B 0,C 180,E1 18625.97,E2 18625.97} C_VEL
LIN {X 0,Y 384.141,Z 1196.234,A -85,B 0,C 180,E1 18622.973,E2 18622.973} C_VEL
LIN {X 0,Y 384.264,Z 1193.368,A -85,B 0,C 180,E1 18619.96,E2 18619.96} C_VEL
LIN {X 0,Y 384.583,Z 1189.469,A -85,B 0,C 180,E1 18616.927,E2 18616.927} C_VEL
LIN {X 0,Y 385.262,Z 1184.517,A -85,B 0,C 180,E1 18613.878,E2 18613.878} C_VEL
LIN {X 0,Y 386.355,Z 1178.475,A -85,B 0,C 180,E1 18610.812,E2 18610.812} C_VEL
LIN {X 0,Y 388.019,Z 1171.181,A -85,B 0,C 180,E1 18607.686,E2 18607.686} C_VEL
LIN {X 0,Y 390.734,Z 1161.225,A -85,B 0,C 180,E1 18604.051,E2 18604.051} C_VEL
LIN {X 0,Y 394.654,Z 1148.618,A -85,B 0,C 180,E1 18600.227,E2 18600.227} C_VEL
LIN {X 0,Y 398.414,Z 1137.629,A -85,B 0,C 180,E1 18597.346,E2 18597.346} C_VEL
LIN {X 0,Y 402.958,Z 1125.194,A -85,B 0,C 180,E1 18594.478,E2 18594.478} C_VEL
LIN {X 0,Y 408.717,Z 1110.004,A -85,B 0,C 180,E1 18591.405,E2 18591.405} C_VEL
LIN {X 0,Y 415.779,Z 1091.588,A -85,B 0,C 180,E1 18588.232,E2 18588.232} C_VEL
LIN {X 0,Y 421.699,Z 1076.234,A -85,B 0,C 180,E1 18585.926,E2 18585.926} C_VEL
LIN {X 0,Y 427.936,Z 1059.894,A -85,B 0,C 180,E1 18583.759,E2 18583.759} C_VEL
LIN {X 0,Y 435.655,Z 1039.29,A -85,B 0,C 180,E1 18581.368,E2 18581.368} C_VEL
LIN {X 0,Y 443.096,Z 1018.126,A -85,B 0,C 180,E1 18579.287,E2 18579.287} C_VEL
LIN {X 0,Y 449.52,Z 998.948,A -85,B 0,C 180,E1 18577.642,E2 18577.642} C_VEL
LIN {X 0,Y 455.748,Z 979.199,A -85,B 0,C 180,E1 18576.162,E2 18576.162} C_VEL
LIN {X 0,Y 463.122,Z 953.857,A -85,B 0,C 180,E1 18574.545,E2 18574.545} C_VEL
LIN {X 0,Y 469.067,Z 930.847,A -85,B 0,C 180,E1 18573.324,E2 18573.324} C_VEL
LIN {X 0,Y 473.984,Z 909.742,A -85,B 0,C 180,E1 18572.375,E2 18572.375} C_VEL
LIN {X 0,Y 478.592,Z 887.336,A -85,B 0,C 180,E1 18571.529,E2 18571.529} C_VEL
LIN {X 0,Y 483.548,Z 858.255,A -85,B 0,C 180,E1 18570.663,E2 18570.663} C_VEL
LIN {X 0,Y 486.653,Z 834.961,A -85,B 0,C 180,E1 18570.136,E2 18570.136} C_VEL
LIN {X 0,Y 488.739,Z 812.312,A -85,B 0,C 180,E1 18569.714,E2 18569.714} C_VEL
LIN {X 0,Y 501.464,Z 595.828,A -85,B 0,C 180,E1 18566.307,E2 18566.307} C_VEL
LIN {X 0,Y 507.943,Z 488.312,A -85,B 0,C 180,E1 18564.604,E2 18564.604} C_VEL
LIN {X 0,Y 497.333,Z 470.99,A -85,B 0,C 180,E1 18561.96,E2 18561.96} C_VEL
LIN {X 0,Y 487.524,Z 455.677,A -85,B 0,C 180,E1 18559.219,E2 18559.219} C_VEL
LIN {X 0,Y 478.4,Z 442.188,A -85,B 0,C 180,E1 18556.327,E2 18556.327} C_VEL
LIN {X 0,Y 470.756,Z 431.525,A -85,B 0,C 180,E1 18553.543,E2 18553.543} C_VEL
LIN {X 0,Y 467.371,Z 426.931,A -85,B 0,C 180,E1 18552.165,E2 18552.165} C_VEL
LIN {X 0,Y 464.273,Z 422.744,A -85,B 0,C 180,E1 18550.799,E2 18550.799} C_VEL
LIN {X 0,Y 460.215,Z 417.292,A -85,B 0,C 180,E1 18548.811,E2 18548.811} C_VEL
LIN {X 0,Y 456.605,Z 412.62,A -85,B 0,C 180,E1 18546.791,E2 18546.791} C_VEL
LIN {X 0,Y 452.873,Z 407.774,A -85,B 0,C 180,E1 18544.305,E2 18544.305} C_VEL
LIN {X 0,Y 448.489,Z 402.148,A -85,B 0,C 180,E1 18540.383,E2 18540.383} C_VEL
LIN {X 0,Y 445.347,Z 398.781,A -85,B 0,C 180,E1 18534.718,E2 18534.718} C_VEL
LIN {X 0,Y 445.237,Z 398.612,A -85,B 0,C 180,E1 18531.606,E2 18531.606} C_VEL
LIN {X 0,Y 446.998,Z 400.844,A -85,B 0,C 180,E1 18527.074,E2 18527.074} C_VEL
LIN {X 0,Y 449.016,Z 402.785,A -85,B 0,C 180,E1 18524.621,E2 18524.621} C_VEL
LIN {X 0,Y 452.617,Z 407.493,A -85,B 0,C 180,E1 18521.451,E2 18521.451} C_VEL
LIN {X 0,Y 454.382,Z 409.921,A -85,B 0,C 180,E1 18520.191,E2 18520.191} C_VEL
LIN {X 0,Y 457.957,Z 414.381,A -85,B 0,C 180,E1 18518.01,E2 18518.01} C_VEL
LIN {X 0,Y 461.8,Z 419.399,A -85,B 0,C 180,E1 18515.98,E2 18515.98} C_VEL
LIN {X 0,Y 465.993,Z 425.048,A -85,B 0,C 180,E1 18514.03,E2 18514.03} C_VEL
LIN {X 0,Y 470.42,Z 431.116,A -85,B 0,C 180,E1 18512.189,E2 18512.189} C_VEL
LIN {X 0,Y 476.076,Z 439.095,A -85,B 0,C 180,E1 18510.078,E2 18510.078} C_VEL
LIN {X 0,Y 484.616,Z 451.538,A -85,B 0,C 180,E1 18507.277,E2 18507.277} C_VEL
LIN {X 0,Y 493.004,Z 464.599,A -85,B 0,C 180,E1 18504.83,E2 18504.83} C_VEL
LIN {X 0,Y 501.963,Z 479.09,A -85,B 0,C 180,E1 18502.479,E2 18502.479} C_VEL
LIN {X 0,Y 503.702,Z 482.28,A -85,B 0,C 180,E1 18502.041,E2 18502.041} C_VEL
LIN {X 0,Y 489.461,Z 714.422,A -85,B 0,C 180,E1 18498.459,E2 18498.459} C_VEL
LIN {X 0,Y 484.594,Z 792.988,A -85,B 0,C 180,E1 18497.221,E2 18497.221} C_VEL
LIN {X 0,Y 481.513,Z 821.428,A -85,B 0,C 180,E1 18496.616,E2 18496.616} C_VEL
LIN {X 0,Y 478.234,Z 843.771,A -85,B 0,C 180,E1 18495.973,E2 18495.973} C_VEL
LIN {X 0,Y 474.704,Z 863.619,A -85,B 0,C 180,E1 18495.275,E2 18495.275} C_VEL
LIN {X 0,Y 469.792,Z 887.271,A -85,B 0,C 180,E1 18494.273,E2 18494.273} C_VEL
LIN {X 0,Y 464.089,Z 910.289,A -85,B 0,C 180,E1 18493.075,E2 18493.075} C_VEL
LIN {X 0,Y 458.553,Z 930.243,A -85,B 0,C 180,E1 18491.853,E2 18491.853} C_VEL
LIN {X 0,Y 452.259,Z 950.949,A -85,B 0,C 180,E1 18490.373,E2 18490.373} C_VEL
LIN {X 0,Y 444.846,Z 972.98,A -85,B 0,C 180,E1 18488.506,E2 18488.506} C_VEL
LIN {X 0,Y 438.473,Z 990.572,A -85,B 0,C 180,E1 18486.768,E2 18486.768} C_VEL
LIN {X 0,Y 431.937,Z 1007.719,A -85,B 0,C 180,E1 18484.827,E2 18484.827} C_VEL
LIN {X 0,Y 424.001,Z 1027.468,A -85,B 0,C 180,E1 18482.204,E2 18482.204} C_VEL
LIN {X 0,Y 417.702,Z 1042.553,A -85,B 0,C 180,E1 18479.86,E2 18479.86} C_VEL
LIN {X 0,Y 411.695,Z 1056.793,A -85,B 0,C 180,E1 18477.323,E2 18477.323} C_VEL
LIN {X 0,Y 405.007,Z 1072.476,A -85,B 0,C 180,E1 18474.038,E2 18474.038} C_VEL
LIN {X 0,Y 400.248,Z 1083.853,A -85,B 0,C 180,E1 18471.237,E2 18471.237} C_VEL
LIN {X 0,Y 395.836,Z 1094.866,A -85,B 0,C 180,E1 18468.101,E2 18468.101} C_VEL
LIN {X 0,Y 391.696,Z 1105.865,A -85,B 0,C 180,E1 18464.336,E2 18464.336} C_VEL
LIN {X 0,Y 389.041,Z 1113.678,A -85,B 0,C 180,E1 18461.113,E2 18461.113} C_VEL
LIN {X 0,Y 387.049,Z 1120.538,A -85,B 0,C 180,E1 18457.72,E2 18457.72} C_VEL
LIN {X 0,Y 385.541,Z 1126.84,A -85,B 0,C 180,E1 18453.717,E2 18453.717} C_VEL
LIN {X 0,Y 384.839,Z 1130.687,A -85,B 0,C 180,E1 18450.446,E2 18450.446} C_VEL
LIN {X 0,Y 384.56,Z 1132.882,A -85,B 0,C 180,E1 18447.962,E2 18447.962} C_VEL
LIN {X 0,Y 383.481,Z 1133.799,A -85,B 0,C 180,E1 18446.823,E2 18446.823} C_VEL
LIN {X 0,Y 376.841,Z 1135.942,A -85,B 0,C 180,E1 18443.523,E2 18443.523} C_VEL
LIN {X 0,Y 376.376,Z 1136.107,A -85,B 0,C 180,E1 18442.762,E2 18442.762} C_VEL
LIN {X 0,Y 376.374,Z 1136.324,A -85,B 0,C 180,E1 18439.593,E2 18439.593} C_VEL
LIN {X 0,Y 376.475,Z 1135.62,A -85,B 0,C 180,E1 18436.484,E2 18436.484} C_VEL
LIN {X 0,Y 376.721,Z 1133.987,A -85,B 0,C 180,E1 18433.343,E2 18433.343} C_VEL
LIN {X 0,Y 377.275,Z 1131.245,A -85,B 0,C 180,E1 18430.009,E2 18430.009} C_VEL
LIN {X 0,Y 378.611,Z 1126.289,A -85,B 0,C 180,E1 18425.837,E2 18425.837} C_VEL
LIN {X 0,Y 380.486,Z 1120.608,A -85,B 0,C 180,E1 18422.281,E2 18422.281} C_VEL
LIN {X 0,Y 382.937,Z 1114.279,A -85,B 0,C 180,E1 18419.044,E2 18419.044} C_VEL
LIN {X 0,Y 386.965,Z 1105.133,A -85,B 0,C 180,E1 18415.178,E2 18415.178} C_VEL
LIN {X 0,Y 391.899,Z 1094.559,A -85,B 0,C 180,E1 18411.562,E2 18411.562} C_VEL
LIN {X 0,Y 397.092,Z 1084.143,A -85,B 0,C 180,E1 18408.53,E2 18408.53} C_VEL
LIN {X 0,Y 404.411,Z 1069.796,A -85,B 0,C 180,E1 18405,E2 18405} C_VEL
LIN {X 0,Y 411.032,Z 1056.802,A -85,B 0,C 180,E1 18402.311,E2 18402.311} C_VEL
LIN {X 0,Y 417.997,Z 1043.032,A -85,B 0,C 180,E1 18399.84,E2 18399.84} C_VEL
LIN {X 0,Y 426.838,Z 1025.179,A -85,B 0,C 180,E1 18397.097,E2 18397.097} C_VEL
LIN {X 0,Y 434.957,Z 1007.8,A -85,B 0,C 180,E1 18394.85,E2 18394.85} C_VEL
LIN {X 0,Y 442.05,Z 991.933,A -85,B 0,C 180,E1 18393.068,E2 18393.068} C_VEL
LIN {X 0,Y 450.109,Z 972.887,A -85,B 0,C 180,E1 18391.215,E2 18391.215} C_VEL
LIN {X 0,Y 458.594,Z 950.827,A -85,B 0,C 180,E1 18389.41,E2 18389.41} C_VEL
LIN {X 0,Y 464.93,Z 932.801,A -85,B 0,C 180,E1 18388.148,E2 18388.148} C_VEL
LIN {X 0,Y 471.185,Z 913.289,A -85,B 0,C 180,E1 18386.97,E2 18386.97} C_VEL
LIN {X 0,Y 478.105,Z 889.055,A -85,B 0,C 180,E1 18385.74,E2 18385.74} C_VEL
LIN {X 0,Y 483.71,Z 865.598,A -85,B 0,C 180,E1 18384.775,E2 18384.775} C_VEL
LIN {X 0,Y 487.78,Z 845.693,A -85,B 0,C 180,E1 18384.099,E2 18384.099} C_VEL
LIN {X 0,Y 491.443,Z 823.989,A -85,B 0,C 180,E1 18383.492,E2 18383.492} C_VEL
LIN {X 0,Y 495.021,Z 795.499,A -85,B 0,C 180,E1 18382.898,E2 18382.898} C_VEL
LIN {X 0,Y 500.374,Z 724.213,A -85,B 0,C 180,E1 18381.776,E2 18381.776} C_VEL
LIN {X 0,Y 517.403,Z 496.538,A -85,B 0,C 180,E1 18378.276,E2 18378.276} C_VEL
LIN {X 0,Y 510.234,Z 484.626,A -85,B 0,C 180,E1 18375.574,E2 18375.574} C_VEL
LIN {X 0,Y 503.961,Z 474.932,A -85,B 0,C 180,E1 18372.781,E2 18372.781} C_VEL
LIN {X 0,Y 500.165,Z 469.28,A -85,B 0,C 180,E1 18370.773,E2 18370.773} C_VEL
LIN {X 0,Y 497.23,Z 464.969,A -85,B 0,C 180,E1 18368.966,E2 18368.966} C_VEL
LIN {X 0,Y 494.969,Z 461.59,A -85,B 0,C 180,E1 18367.312,E2 18367.312} C_VEL
LIN {X 0,Y 491.812,Z 456.892,A -85,B 0,C 180,E1 18364.314,E2 18364.314} C_VEL
LIN {X 0,Y 489.145,Z 453.216,A -85,B 0,C 180,E1 18359.063,E2 18359.063} C_VEL
LIN {X 0,Y 489.183,Z 453.284,A -85,B 0,C 180,E1 18356.484,E2 18356.484} C_VEL
LIN {X 0,Y 492.184,Z 457.28,A -85,B 0,C 180,E1 18351,E2 18351} C_VEL
LIN {X 0,Y 496.094,Z 463.234,A -85,B 0,C 180,E1 18347.546,E2 18347.546} C_VEL
LIN {X 0,Y 499.563,Z 468.478,A -85,B 0,C 180,E1 18345.274,E2 18345.274} C_VEL
LIN {X 0,Y 502.51,Z 472.917,A -85,B 0,C 180,E1 18343.647,E2 18343.647} C_VEL
LIN {X 0,Y 507.723,Z 480.742,A -85,B 0,C 180,E1 18341.187,E2 18341.187} C_VEL
LIN {X 0,Y 514.686,Z 492.061,A -85,B 0,C 180,E1 18338.399,E2 18338.399} C_VEL
LIN {X 0,Y 518.958,Z 499.646,A -85,B 0,C 180,E1 18336.876,E2 18336.876} C_VEL
LIN {X 0,Y 502.796,Z 717.619,A -85,B 0,C 180,E1 18333.424,E2 18333.424} C_VEL
LIN {X 0,Y 495.591,Z 816.265,A -85,B 0,C 180,E1 18331.842,E2 18331.842} C_VEL
LIN {X 0,Y 492.096,Z 844.618,A -85,B 0,C 180,E1 18331.289,E2 18331.289} C_VEL
LIN {X 0,Y 487.828,Z 868.979,A -85,B 0,C 180,E1 18330.68,E2 18330.68} C_VEL
LIN {X 0,Y 483.388,Z 890.238,A -85,B 0,C 180,E1 18330.015,E2 18330.015} C_VEL
LIN {X 0,Y 478.06,Z 912.367,A -85,B 0,C 180,E1 18329.174,E2 18329.174} C_VEL
LIN {X 0,Y 470.581,Z 939.37,A -85,B 0,C 180,E1 18327.913,E2 18327.913} C_VEL
LIN {X 0,Y 463.725,Z 961.144,A -85,B 0,C 180,E1 18326.679,E2 18326.679} C_VEL
LIN {X 0,Y 456.931,Z 981.029,A -85,B 0,C 180,E1 18325.362,E2 18325.362} C_VEL
LIN {X 0,Y 449.914,Z 1000.232,A -85,B 0,C 180,E1 18323.894,E2 18323.894} C_VEL
LIN {X 0,Y 441.048,Z 1022.958,A -85,B 0,C 180,E1 18321.874,E2 18321.874} C_VEL
LIN {X 0,Y 432.506,Z 1043.415,A -85,B 0,C 180,E1 18319.719,E2 18319.719} C_VEL
LIN {X 0,Y 425.5,Z 1059.732,A -85,B 0,C 180,E1 18317.749,E2 18317.749} C_VEL
LIN {X 0,Y 418.537,Z 1075.607,A -85,B 0,C 180,E1 18315.574,E2 18315.574} C_VEL
LIN {X 0,Y 410.683,Z 1093.444,A -85,B 0,C 180,E1 18312.786,E2 18312.786} C_VEL
LIN {X 0,Y 403.021,Z 1110.718,A -85,B 0,C 180,E1 18309.613,E2 18309.613} C_VEL
LIN {X 0,Y 397.295,Z 1124.06,A -85,B 0,C 180,E1 18306.796,E2 18306.796} C_VEL
LIN {X 0,Y 392.116,Z 1136.682,A -85,B 0,C 180,E1 18303.767,E2 18303.767} C_VEL
LIN {X 0,Y 386.971,Z 1150.2,A -85,B 0,C 180,E1 18300.048,E2 18300.048} C_VEL
LIN {X 0,Y 382.909,Z 1161.944,A -85,B 0,C 180,E1 18296.187,E2 18296.187} C_VEL
LIN {X 0,Y 380.351,Z 1170.553,A -85,B 0,C 180,E1 18292.896,E2 18292.896} C_VEL
LIN {X 0,Y 378.605,Z 1177.622,A -85,B 0,C 180,E1 18289.757,E2 18289.757} C_VEL
LIN {X 0,Y 377.33,Z 1184.002,A -85,B 0,C 180,E1 18286.408,E2 18286.408} C_VEL
LIN {X 0,Y 376.57,Z 1189.351,A -85,B 0,C 180,E1 18282.971,E2 18282.971} C_VEL
LIN {X 0,Y 376.209,Z 1194.021,A -85,B 0,C 180,E1 18279.022,E2 18279.022} C_VEL
LIN {X 0,Y 376.154,Z 1196.794,A -85,B 0,C 180,E1 18275.338,E2 18275.338} C_VEL
LIN {X 0,Y 376.172,Z 1198.082,A -85,B 0,C 180,E1 18272.133,E2 18272.133} C_VEL
LIN {X 0,Y 376.172,Z 1198.289,A -85,B 0,C 180,E1 18269.086,E2 18269.086} C_VEL
LIN {X 0,Y 376.154,Z 1197.487,A -85,B 0,C 180,E1 18266.037,E2 18266.037} C_VEL
LIN {X 0,Y 376.16,Z 1195.673,A -85,B 0,C 180,E1 18262.977,E2 18262.977} C_VEL
LIN {X 0,Y 376.28,Z 1192.84,A -85,B 0,C 180,E1 18259.9,E2 18259.9} C_VEL
LIN {X 0,Y 376.61,Z 1188.969,A -85,B 0,C 180,E1 18256.802,E2 18256.802} C_VEL
LIN {X 0,Y 377.306,Z 1184.042,A -85,B 0,C 180,E1 18253.686,E2 18253.686} C_VEL
LIN {X 0,Y 378.456,Z 1178.03,A -85,B 0,C 180,E1 18250.556,E2 18250.556} C_VEL
LIN {X 0,Y 380.163,Z 1170.836,A -85,B 0,C 180,E1 18247.397,E2 18247.397} C_VEL
LIN {X 0,Y 382.723,Z 1161.761,A -85,B 0,C 180,E1 18243.991,E2 18243.991} C_VEL
LIN {X 0,Y 386.921,Z 1148.809,A -85,B 0,C 180,E1 18239.913,E2 18239.913} C_VEL
LIN {X 0,Y 391.034,Z 1137.29,A -85,B 0,C 180,E1 18236.826,E2 18236.826} C_VEL
LIN {X 0,Y 395.644,Z 1125.152,A -85,B 0,C 180,E1 18233.971,E2 18233.971} C_VEL
LIN {X 0,Y 401.206,Z 1110.97,A -85,B 0,C 180,E1 18231.039,E2 18231.039} C_VEL
LIN {X 0,Y 408.694,Z 1092.236,A -85,B 0,C 180,E1 18227.718,E2 18227.718} C_VEL
LIN {X 0,Y 415.207,Z 1075.924,A -85,B 0,C 180,E1 18225.231,E2 18225.231} C_VEL
LIN {X 0,Y 421.561,Z 1059.831,A -85,B 0,C 180,E1 18223.071,E2 18223.071} C_VEL
LIN {X 0,Y 429.388,Z 1039.585,A -85,B 0,C 180,E1 18220.694,E2 18220.694} C_VEL
LIN {X 0,Y 437.234,Z 1018.022,A -85,B 0,C 180,E1 18218.549,E2 18218.549} C_VEL
LIN {X 0,Y 443.575,Z 999.652,A -85,B 0,C 180,E1 18216.958,E2 18216.958} C_VEL
LIN {X 0,Y 449.68,Z 980.871,A -85,B 0,C 180,E1 18215.532,E2 18215.532} C_VEL
LIN {X 0,Y 456.107,Z 959.736,A -85,B 0,C 180,E1 18214.14,E2 18214.14} C_VEL
LIN {X 0,Y 463.296,Z 933.37,A -85,B 0,C 180,E1 18212.683,E2 18212.683} C_VEL
LIN {X 0,Y 468.538,Z 911.614,A -85,B 0,C 180,E1 18211.687,E2 18211.687} C_VEL
LIN {X 0,Y 472.998,Z 890.722,A -85,B 0,C 180,E1 18210.882,E2 18210.882} C_VEL
LIN {X 0,Y 477.286,Z 867.545,A -85,B 0,C 180,E1 18210.146,E2 18210.146} C_VEL
LIN {X 0,Y 481.59,Z 838.172,A -85,B 0,C 180,E1 18209.431,E2 18209.431} C_VEL
LIN {X 0,Y 483.907,Z 814.938,A -85,B 0,C 180,E1 18208.988,E2 18208.988} C_VEL
LIN {X 0,Y 496.594,Z 605.967,A -85,B 0,C 180,E1 18205.684,E2 18205.684} C_VEL
LIN {X 0,Y 503.637,Z 492.67,A -85,B 0,C 180,E1 18203.892,E2 18203.892} C_VEL
LIN {X 0,Y 493.574,Z 476.018,A -85,B 0,C 180,E1 18201.293,E2 18201.293} C_VEL
LIN {X 0,Y 484.361,Z 461.536,A -85,B 0,C 180,E1 18198.63,E2 18198.63} C_VEL
LIN {X 0,Y 476.032,Z 449.061,A -85,B 0,C 180,E1 18195.909,E2 18195.909} C_VEL
LIN {X 0,Y 468.766,Z 438.73,A -85,B 0,C 180,E1 18193.193,E2 18193.193} C_VEL
LIN {X 0,Y 463.266,Z 430.997,A -85,B 0,C 180,E1 18190.823,E2 18190.823} C_VEL
LIN {X 0,Y 458.504,Z 424.677,A -85,B 0,C 180,E1 18188.465,E2 18188.465} C_VEL
LIN {X 0,Y 455.187,Z 420.284,A -85,B 0,C 180,E1 18186.559,E2 18186.559} C_VEL
LIN {X 0,Y 451.53,Z 415.479,A -85,B 0,C 180,E1 18184.064,E2 18184.064} C_VEL
LIN {X 0,Y 447.39,Z 410.02,A -85,B 0,C 180,E1 18180.256,E2 18180.256} C_VEL
LIN {X 0,Y 444.342,Z 406.679,A -85,B 0,C 180,E1 18174.577,E2 18174.577} C_VEL
LIN {X 0,Y 444.28,Z 406.579,A -85,B 0,C 180,E1 18171.458,E2 18171.458} C_VEL
LIN {X 0,Y 446.31,Z 409.096,A -85,B 0,C 180,E1 18166.658,E2 18166.658} C_VEL
LIN {X 0,Y 447.871,Z 410.59,A -85,B 0,C 180,E1 18164.792,E2 18164.792} C_VEL
LIN {X 0,Y 451.328,Z 415.237,A -85,B 0,C 180,E1 18161.664,E2 18161.664} C_VEL
LIN {X 0,Y 452.917,Z 417.418,A -85,B 0,C 180,E1 18160.5,E2 18160.5} C_VEL
LIN {X 0,Y 456.678,Z 422.264,A -85,B 0,C 180,E1 18158.148,E2 18158.148} C_VEL
LIN {X 0,Y 460.235,Z 426.984,A -85,B 0,C 180,E1 18156.233,E2 18156.233} C_VEL
LIN {X 0,Y 464.48,Z 432.813,A -85,B 0,C 180,E1 18154.224,E2 18154.224} C_VEL
LIN {X 0,Y 468.811,Z 438.829,A -85,B 0,C 180,E1 18152.396,E2 18152.396} C_VEL
LIN {X 0,Y 475.977,Z 449.075,A -85,B 0,C 180,E1 18149.723,E2 18149.723} C_VEL
LIN {X 0,Y 485.332,Z 463.254,A -85,B 0,C 180,E1 18146.698,E2 18146.698} C_VEL
LIN {X 0,Y 495.685,Z 479.953,A -85,B 0,C 180,E1 18143.769,E2 18143.769} C_VEL
LIN {X 0,Y 499.477,Z 486.596,A -85,B 0,C 180,E1 18142.773,E2 18142.773} C_VEL
LIN {X 0,Y 484.807,Z 719.193,A -85,B 0,C 180,E1 18139.177,E2 18139.177} C_VEL
LIN {X 0,Y 480.056,Z 793.478,A -85,B 0,C 180,E1 18138.002,E2 18138.002} C_VEL
LIN {X 0,Y 476.857,Z 822.207,A -85,B 0,C 180,E1 18137.389,E2 18137.389} C_VEL
LIN {X 0,Y 473.538,Z 844.3,A -85,B 0,C 180,E1 18136.751,E2 18136.751} C_VEL
LIN {X 0,Y 470.009,Z 863.69,A -85,B 0,C 180,E1 18136.071,E2 18136.071} C_VEL
LIN {X 0,Y 464.855,Z 887.954,A -85,B 0,C 180,E1 18135.044,E2 18135.044} C_VEL
LIN {X 0,Y 459.006,Z 910.928,A -85,B 0,C 180,E1 18133.844,E2 18133.844} C_VEL
LIN {X 0,Y 453.329,Z 930.869,A -85,B 0,C 180,E1 18132.619,E2 18132.619} C_VEL
LIN {X 0,Y 446.644,Z 952.291,A -85,B 0,C 180,E1 18131.08,E2 18131.08} C_VEL
LIN {X 0,Y 439.013,Z 974.244,A -85,B 0,C 180,E1 18129.198,E2 18129.198} C_VEL
LIN {X 0,Y 432.465,Z 991.773,A -85,B 0,C 180,E1 18127.449,E2 18127.449} C_VEL
LIN {X 0,Y 425.123,Z 1010.459,A -85,B 0,C 180,E1 18125.299,E2 18125.299} C_VEL
LIN {X 0,Y 417.272,Z 1029.203,A -85,B 0,C 180,E1 18122.745,E2 18122.745} C_VEL
LIN {X 0,Y 411.231,Z 1043.19,A -85,B 0,C 180,E1 18120.541,E2 18120.541} C_VEL
LIN {X 0,Y 405.005,Z 1057.428,A -85,B 0,C 180,E1 18117.973,E2 18117.973} C_VEL
LIN {X 0,Y 398.057,Z 1073.118,A -85,B 0,C 180,E1 18114.643,E2 18114.643} C_VEL
LIN {X 0,Y 393.093,Z 1084.499,A -85,B 0,C 180,E1 18111.799,E2 18111.799} C_VEL
LIN {X 0,Y 388.489,Z 1095.509,A -85,B 0,C 180,E1 18108.611,E2 18108.611} C_VEL
LIN {X 0,Y 384.148,Z 1106.513,A -85,B 0,C 180,E1 18104.778,E2 18104.778} C_VEL
LIN {X 0,Y 381.465,Z 1113.999,A -85,B 0,C 180,E1 18101.644,E2 18101.644} C_VEL
LIN {X 0,Y 379.391,Z 1120.622,A -85,B 0,C 180,E1 18098.334,E2 18098.334} C_VEL
LIN {X 0,Y 377.74,Z 1127.105,A -85,B 0,C 180,E1 18094.25,E2 18094.25} C_VEL
LIN {X 0,Y 376.929,Z 1131.188,A -85,B 0,C 180,E1 18090.76,E2 18090.76} C_VEL
LIN {X 0,Y 376.567,Z 1133.781,A -85,B 0,C 180,E1 18087.717,E2 18087.717} C_VEL
LIN {X 0,Y 376.401,Z 1135.479,A -85,B 0,C 180,E1 18084.665,E2 18084.665} C_VEL
LIN {X 0,Y 376.376,Z 1136.107,A -85,B 0,C 180,E1 18082.762,E2 18082.762} C_VEL
LIN {X 0,Y 375.358,Z 1136.373,A -85,B 0,C 180,E1 18081.59,E2 18081.59} C_VEL
LIN {X 0,Y 368.987,Z 1136.912,A -85,B 0,C 180,E1 18078.279,E2 18078.279} C_VEL
LIN {X 0,Y 368.477,Z 1136.697,A -85,B 0,C 180,E1 18077.415,E2 18077.415} C_VEL
LIN {X 0,Y 368.731,Z 1134.976,A -85,B 0,C 180,E1 18073.62,E2 18073.62} C_VEL
LIN {X 0,Y 369.244,Z 1132.526,A -85,B 0,C 180,E1 18070.38,E2 18070.38} C_VEL
LIN {X 0,Y 370.165,Z 1129.057,A -85,B 0,C 180,E1 18067.09,E2 18067.09} C_VEL
LIN {X 0,Y 372.116,Z 1123.365,A -85,B 0,C 180,E1 18062.993,E2 18062.993} C_VEL
LIN {X 0,Y 375.007,Z 1116.041,A -85,B 0,C 180,E1 18059.03,E2 18059.03} C_VEL
LIN {X 0,Y 378.32,Z 1108.69,A -85,B 0,C 180,E1 18055.741,E2 18055.741} C_VEL
LIN {X 0,Y 383.509,Z 1098.211,A -85,B 0,C 180,E1 18051.838,E2 18051.838} C_VEL
LIN {X 0,Y 389.44,Z 1086.649,A -85,B 0,C 180,E1 18048.32,E2 18048.32} C_VEL
LIN {X 0,Y 395.527,Z 1075.22,A -85,B 0,C 180,E1 18045.351,E2 18045.351} C_VEL
LIN {X 0,Y 404.071,Z 1059.22,A -85,B 0,C 180,E1 18041.857,E2 18041.857} C_VEL
LIN {X 0,Y 411.205,Z 1045.637,A -85,B 0,C 180,E1 18039.355,E2 18039.355} C_VEL
LIN {X 0,Y 418.546,Z 1031.356,A -85,B 0,C 180,E1 18037.071,E2 18037.071} C_VEL
LIN {X 0,Y 428.049,Z 1012.19,A -85,B 0,C 180,E1 18034.456,E2 18034.456} C_VEL
LIN {X 0,Y 436.162,Z 994.674,A -85,B 0,C 180,E1 18032.442,E2 18032.442} C_VEL
LIN {X 0,Y 443.429,Z 978.078,A -85,B 0,C 180,E1 18030.785,E2 18030.785} C_VEL
LIN {X 0,Y 451.742,Z 957.818,A -85,B 0,C 180,E1 18029.041,E2 18029.041} C_VEL
LIN {X 0,Y 460.083,Z 935.081,A -85,B 0,C 180,E1 18027.407,E2 18027.407} C_VEL
LIN {X 0,Y 466.7,Z 915.07,A -85,B 0,C 180,E1 18026.19,E2 18026.19} C_VEL
LIN {X 0,Y 473.065,Z 893.64,A -85,B 0,C 180,E1 18025.087,E2 18025.087} C_VEL
LIN {X 0,Y 479.444,Z 868.327,A -85,B 0,C 180,E1 18024.017,E2 18024.017} C_VEL
LIN {X 0,Y 483.819,Z 847.659,A -85,B 0,C 180,E1 18023.306,E2 18023.306} C_VEL
LIN {X 0,Y 487.483,Z 826.714,A -85,B 0,C 180,E1 18022.711,E2 18022.711} C_VEL
LIN {X 0,Y 491.111,Z 800.353,A -85,B 0,C 180,E1 18022.139,E2 18022.139} C_VEL
LIN {X 0,Y 494.745,Z 755.462,A -85,B 0,C 180,E1 18021.419,E2 18021.419} C_VEL
LIN {X 0,Y 512.957,Z 516.773,A -85,B 0,C 180,E1 18017.752,E2 18017.752} C_VEL
LIN {X 0,Y 514.132,Z 501.669,A -85,B 0,C 180,E1 18017.515,E2 18017.515} C_VEL
LIN {X 0,Y 507.906,Z 491.178,A -85,B 0,C 180,E1 18015.062,E2 18015.062} C_VEL
LIN {X 0,Y 502.177,Z 482.157,A -85,B 0,C 180,E1 18012.418,E2 18012.418} C_VEL
LIN {X 0,Y 498.683,Z 476.819,A -85,B 0,C 180,E1 18010.513,E2 18010.513} C_VEL
LIN {X 0,Y 495.736,Z 472.399,A -85,B 0,C 180,E1 18008.642,E2 18008.642} C_VEL
LIN {X 0,Y 493.824,Z 469.448,A -85,B 0,C 180,E1 18007.199,E2 18007.199} C_VEL
LIN {X 0,Y 490.729,Z 464.77,A -85,B 0,C 180,E1 18004.207,E2 18004.207} C_VEL
LIN {X 0,Y 488.166,Z 461.163,A -85,B 0,C 180,E1 17999.061,E2 17999.061} C_VEL
LIN {X 0,Y 488.186,Z 461.189,A -85,B 0,C 180,E1 17996.595,E2 17996.595} C_VEL
LIN {X 0,Y 491.094,Z 465.17,A -85,B 0,C 180,E1 17991.098,E2 17991.098} C_VEL
LIN {X 0,Y 494.868,Z 471.056,A -85,B 0,C 180,E1 17987.692,E2 17987.692} C_VEL
LIN {X 0,Y 498.191,Z 476.18,A -85,B 0,C 180,E1 17985.47,E2 17985.47} C_VEL
LIN {X 0,Y 501.082,Z 480.642,A -85,B 0,C 180,E1 17983.837,E2 17983.837} C_VEL
LIN {X 0,Y 505.969,Z 488.115,A -85,B 0,C 180,E1 17981.478,E2 17981.478} C_VEL
LIN {X 0,Y 512.658,Z 499.213,A -85,B 0,C 180,E1 17978.729,E2 17978.729} C_VEL
LIN {X 0,Y 515.627,Z 504.676,A -85,B 0,C 180,E1 17977.625,E2 17977.625} C_VEL
LIN {X 0,Y 498.931,Z 724.067,A -85,B 0,C 180,E1 17974.156,E2 17974.156} C_VEL
LIN {X 0,Y 491.997,Z 816.096,A -85,B 0,C 180,E1 17972.678,E2 17972.678} C_VEL
LIN {X 0,Y 488.351,Z 844.802,A -85,B 0,C 180,E1 17972.117,E2 17972.117} C_VEL
LIN {X 0,Y 484.044,Z 868.821,A -85,B 0,C 180,E1 17971.521,E2 17971.521} C_VEL
LIN {X 0,Y 479.589,Z 889.689,A -85,B 0,C 180,E1 17970.873,E2 17970.873} C_VEL
LIN {X 0,Y 474.241,Z 911.377,A -85,B 0,C 180,E1 17970.057,E2 17970.057} C_VEL
LIN {X 0,Y 467.107,Z 936.79,A -85,B 0,C 180,E1 17968.894,E2 17968.894} C_VEL
LIN {X 0,Y 459.558,Z 960.206,A -85,B 0,C 180,E1 17967.583,E2 17967.583} C_VEL
LIN {X 0,Y 452.607,Z 980.049,A -85,B 0,C 180,E1 17966.277,E2 17966.277} C_VEL
LIN {X 0,Y 445.624,Z 998.598,A -85,B 0,C 180,E1 17964.869,E2 17964.869} C_VEL
LIN {X 0,Y 436.769,Z 1020.788,A -85,B 0,C 180,E1 17962.92,E2 17962.92} C_VEL
LIN {X 0,Y 427.642,Z 1041.947,A -85,B 0,C 180,E1 17960.706,E2 17960.706} C_VEL
LIN {X 0,Y 420.046,Z 1058.993,A -85,B 0,C 180,E1 17958.646,E2 17958.646} C_VEL
LIN {X 0,Y 412.686,Z 1075.149,A -85,B 0,C 180,E1 17956.421,E2 17956.421} C_VEL
LIN {X 0,Y 404.119,Z 1093.855,A -85,B 0,C 180,E1 17953.458,E2 17953.458} C_VEL
LIN {X 0,Y 396.168,Z 1110.953,A -85,B 0,C 180,E1 17950.248,E2 17950.248} C_VEL
LIN {X 0,Y 390.215,Z 1124.204,A -85,B 0,C 180,E1 17947.393,E2 17947.393} C_VEL
LIN {X 0,Y 384.755,Z 1136.922,A -85,B 0,C 180,E1 17944.268,E2 17944.268} C_VEL
LIN {X 0,Y 378.873,Z 1151.623,A -85,B 0,C 180,E1 17940.045,E2 17940.045} C_VEL
LIN {X 0,Y 375.217,Z 1161.777,A -85,B 0,C 180,E1 17936.595,E2 17936.595} C_VEL
LIN {X 0,Y 372.651,Z 1169.942,A -85,B 0,C 180,E1 17933.397,E2 17933.397} C_VEL
LIN {X 0,Y 370.793,Z 1176.998,A -85,B 0,C 180,E1 17930.191,E2 17930.191} C_VEL
LIN {X 0,Y 369.439,Z 1183.262,A -85,B 0,C 180,E1 17926.833,E2 17926.833} C_VEL
LIN {X 0,Y 368.661,Z 1188.384,A -85,B 0,C 180,E1 17923.488,E2 17923.488} C_VEL
LIN {X 0,Y 368.25,Z 1193.085,A -85,B 0,C 180,E1 17919.534,E2 17919.534} C_VEL
LIN {X 0,Y 368.171,Z 1196.066,A -85,B 0,C 180,E1 17915.611,E2 17915.611} C_VEL
LIN {X 0,Y 368.197,Z 1197.4,A -85,B 0,C 180,E1 17912.335,E2 17912.335} C_VEL
LIN {X 0,Y 368.195,Z 1197.648,A -85,B 0,C 180,E1 17909.222,E2 17909.222} C_VEL
LIN {X 0,Y 368.179,Z 1196.886,A -85,B 0,C 180,E1 17906.107,E2 17906.107} C_VEL
LIN {X 0,Y 368.188,Z 1194.984,A -85,B 0,C 180,E1 17902.824,E2 17902.824} C_VEL
LIN {X 0,Y 368.308,Z 1192.13,A -85,B 0,C 180,E1 17899.679,E2 17899.679} C_VEL
LIN {X 0,Y 368.667,Z 1188.24,A -85,B 0,C 180,E1 17896.512,E2 17896.512} C_VEL
LIN {X 0,Y 369.399,Z 1183.286,A -85,B 0,C 180,E1 17893.327,E2 17893.327} C_VEL
LIN {X 0,Y 370.64,Z 1177.243,A -85,B 0,C 180,E1 17890.129,E2 17890.129} C_VEL
LIN {X 0,Y 372.424,Z 1170.07,A -85,B 0,C 180,E1 17886.923,E2 17886.923} C_VEL
LIN {X 0,Y 375.035,Z 1161.279,A -85,B 0,C 180,E1 17883.562,E2 17883.562} C_VEL
LIN {X 0,Y 379.391,Z 1148.441,A -85,B 0,C 180,E1 17879.427,E2 17879.427} C_VEL
LIN {X 0,Y 383.924,Z 1136.322,A -85,B 0,C 180,E1 17876.129,E2 17876.129} C_VEL
LIN {X 0,Y 388.808,Z 1123.965,A -85,B 0,C 180,E1 17873.189,E2 17873.189} C_VEL
LIN {X 0,Y 395.103,Z 1108.635,A -85,B 0,C 180,E1 17870.001,E2 17870.001} C_VEL
LIN {X 0,Y 402.38,Z 1091.071,A -85,B 0,C 180,E1 17866.895,E2 17866.895} C_VEL
LIN {X 0,Y 408.767,Z 1075.636,A -85,B 0,C 180,E1 17864.519,E2 17864.519} C_VEL
LIN {X 0,Y 415.304,Z 1059.611,A -85,B 0,C 180,E1 17862.344,E2 17862.344} C_VEL
LIN {X 0,Y 422.73,Z 1040.965,A -85,B 0,C 180,E1 17860.125,E2 17860.125} C_VEL
LIN {X 0,Y 431.444,Z 1017.894,A -85,B 0,C 180,E1 17857.791,E2 17857.791} C_VEL
LIN {X 0,Y 438.093,Z 999.185,A -85,B 0,C 180,E1 17856.163,E2 17856.163} C_VEL
LIN {X 0,Y 444.609,Z 979.669,A -85,B 0,C 180,E1 17854.679,E2 17854.679} C_VEL
LIN {X 0,Y 452.06,Z 955.7,A -85,B 0,C 180,E1 17853.116,E2 17853.116} C_VEL
LIN {X 0,Y 458.781,Z 931.093,A -85,B 0,C 180,E1 17851.793,E2 17851.793} C_VEL
LIN {X 0,Y 463.977,Z 909.912,A -85,B 0,C 180,E1 17850.835,E2 17850.835} C_VEL
LIN {X 0,Y 468.579,Z 888.7,A -85,B 0,C 180,E1 17850.028,E2 17850.028} C_VEL
LIN {X 0,Y 473.53,Z 862.088,A -85,B 0,C 180,E1 17849.206,E2 17849.206} C_VEL
LIN {X 0,Y 477.28,Z 835.585,A -85,B 0,C 180,E1 17848.595,E2 17848.595} C_VEL
LIN {X 0,Y 479.491,Z 813.158,A -85,B 0,C 180,E1 17848.172,E2 17848.172} C_VEL
LIN {X 0,Y 492.78,Z 600.301,A -85,B 0,C 180,E1 17844.801,E2 17844.801} C_VEL
LIN {X 0,Y 499.344,Z 496.923,A -85,B 0,C 180,E1 17843.152,E2 17843.152} C_VEL
LIN {X 0,Y 490.16,Z 481.601,A -85,B 0,C 180,E1 17840.697,E2 17840.697} C_VEL
LIN {X 0,Y 481.34,Z 467.505,A -85,B 0,C 180,E1 17838.062,E2 17838.062} C_VEL
LIN {X 0,Y 473.289,Z 455.361,A -85,B 0,C 180,E1 17835.344,E2 17835.344} C_VEL
LIN {X 0,Y 466.512,Z 445.512,A -85,B 0,C 180,E1 17832.722,E2 17832.722} C_VEL
LIN {X 0,Y 461.075,Z 437.907,A -85,B 0,C 180,E1 17830.306,E2 17830.306} C_VEL
LIN {X 0,Y 457.034,Z 432.331,A -85,B 0,C 180,E1 17828.239,E2 17828.239} C_VEL
LIN {X 0,Y 453.776,Z 427.948,A -85,B 0,C 180,E1 17826.325,E2 17826.325} C_VEL
LIN {X 0,Y 450.195,Z 423.182,A -85,B 0,C 180,E1 17823.82,E2 17823.82} C_VEL
LIN {X 0,Y 446.292,Z 417.891,A -85,B 0,C 180,E1 17820.128,E2 17820.128} C_VEL
LIN {X 0,Y 443.361,Z 414.622,A -85,B 0,C 180,E1 17814.565,E2 17814.565} C_VEL
LIN {X 0,Y 443.305,Z 414.526,A -85,B 0,C 180,E1 17811.439,E2 17811.439} C_VEL
LIN {X 0,Y 445.449,Z 417.165,A -85,B 0,C 180,E1 17806.5,E2 17806.5} C_VEL
LIN {X 0,Y 446.794,Z 418.521,A -85,B 0,C 180,E1 17804.887,E2 17804.887} C_VEL
LIN {X 0,Y 450.214,Z 423.137,A -85,B 0,C 180,E1 17801.751,E2 17801.751} C_VEL
LIN {X 0,Y 455.193,Z 429.84,A -85,B 0,C 180,E1 17798.412,E2 17798.412} C_VEL
LIN {X 0,Y 458.679,Z 434.567,A -85,B 0,C 180,E1 17796.489,E2 17796.489} C_VEL
LIN {X 0,Y 462.726,Z 440.212,A -85,B 0,C 180,E1 17794.531,E2 17794.531} C_VEL
LIN {X 0,Y 468.497,Z 448.258,A -85,B 0,C 180,E1 17792.09,E2 17792.09} C_VEL
LIN {X 0,Y 477.144,Z 461.218,A -85,B 0,C 180,E1 17788.933,E2 17788.933} C_VEL
LIN {X 0,Y 485.68,Z 474.718,A -85,B 0,C 180,E1 17786.23,E2 17786.23} C_VEL
LIN {X 0,Y 494.717,Z 489.696,A -85,B 0,C 180,E1 17783.687,E2 17783.687} C_VEL
LIN {X 0,Y 495.324,Z 491.034,A -85,B 0,C 180,E1 17783.516,E2 17783.516} C_VEL
LIN {X 0,Y 480.23,Z 723.954,A -85,B 0,C 180,E1 17779.909,E2 17779.909} C_VEL
LIN {X 0,Y 475.6,Z 794.068,A -85,B 0,C 180,E1 17778.795,E2 17778.795} C_VEL
LIN {X 0,Y 472.289,Z 822.966,A -85,B 0,C 180,E1 17778.176,E2 17778.176} C_VEL
LIN {X 0,Y 468.91,Z 844.899,A -85,B 0,C 180,E1 17777.542,E2 17777.542} C_VEL
LIN {X 0,Y 465.251,Z 864.494,A -85,B 0,C 180,E1 17776.853,E2 17776.853} C_VEL
LIN {X 0,Y 460,Z 888.601,A -85,B 0,C 180,E1 17775.831,E2 17775.831} C_VEL
LIN {X 0,Y 454.008,Z 911.56,A -85,B 0,C 180,E1 17774.63,E2 17774.63} C_VEL
LIN {X 0,Y 448.449,Z 930.643,A -85,B 0,C 180,E1 17773.458,E2 17773.458} C_VEL
LIN {X 0,Y 442.057,Z 950.658,A -85,B 0,C 180,E1 17772.028,E2 17772.028} C_VEL
LIN {X 0,Y 433.719,Z 974.216,A -85,B 0,C 180,E1 17770.029,E2 17770.029} C_VEL
LIN {X 0,Y 426.972,Z 991.815,A -85,B 0,C 180,E1 17768.271,E2 17768.271} C_VEL
